LIN {X 0,Y 247.063,Z 768.988,A -85,B 0,C 180,E1 -18816.531,E2 -18816.531} C_VEL
LIN {X 0,Y 247.331,Z 765.214,A -85,B 0,C 180,E1 -18819.814,E2 -18819.814} C_VEL
LIN {X 0,Y 248.197,Z 759.827,A -85,B 0,C 180,E1 -18823.091,E2 -18823.091} C_VEL
LIN {X 0,Y 249.368,Z 753.588,A -85,B 0,C 180,E1 -18825.947,E2 -18825.947} C_VEL
LIN {X 0,Y 251.192,Z 745.733,A -85,B 0,C 180,E1 -18828.767,E2 -18828.767} C_VEL
LIN {X 0,Y 253.14,Z 737.491,A -85,B 0,C 180,E1 -18831.154,E2 -18831.154} C_VEL
LIN {X 0,Y 255.134,Z 729.322,A -85,B 0,C 180,E1 -18833.11,E2 -18833.11} C_VEL
LIN {X 0,Y 257.768,Z 718.537,A -85,B 0,C 180,E1 -18835.212,E2 -18835.212} C_VEL
LIN {X 0,Y 260.138,Z 707.083,A -85,B 0,C 180,E1 -18837.029,E2 -18837.029} C_VEL
LIN {X 0,Y 262.65,Z 694.698,A -85,B 0,C 180,E1 -18838.572,E2 -18838.572} C_VEL
LIN {X 0,Y 264.885,Z 681.638,A -85,B 0,C 180,E1 -18839.831,E2 -18839.831} C_VEL
LIN {X 0,Y 266.701,Z 667.987,A -85,B 0,C 180,E1 -18840.808,E2 -18840.808} C_VEL
LIN {X 0,Y 268.128,Z 653.813,A -85,B 0,C 180,E1 -18841.503,E2 -18841.503} C_VEL
LIN {X 0,Y 269.125,Z 632.659,A -85,B 0,C 180,E1 -18842.143,E2 -18842.143} C_VEL
LIN {X 0,Y 271.804,Z 565.547,A -85,B 0,C 180,E1 -18843.958,E2 -18843.958} C_VEL
LIN {X 0,Y 269.236,Z 545.201,A -85,B 0,C 180,E1 -18844.967,E2 -18844.967} C_VEL
LIN {X 0,Y 261.457,Z 528.213,A -85,B 0,C 180,E1 -18846.671,E2 -18846.671} C_VEL
LIN {X 0,Y 257.903,Z 520.842,A -85,B 0,C 180,E1 -18847.537,E2 -18847.537} C_VEL
LIN {X 0,Y 255.154,Z 510.348,A -85,B 0,C 180,E1 -18851.377,E2 -18851.377} C_VEL
LIN {X 0,Y 252.343,Z 500.973,A -85,B 0,C 180,E1 -18855.158,E2 -18855.158} C_VEL
LIN {X 0,Y 249.727,Z 493.237,A -85,B 0,C 180,E1 -18858.597,E2 -18858.597} C_VEL
LIN {X 0,Y 249.076,Z 491.075,A -85,B 0,C 180,E1 -18859.623,E2 -18859.623} C_VEL
LIN {X 0,Y 249.067,Z 491.051,A -85,B 0,C 180,E1 -18863.661,E2 -18863.661} C_VEL
LIN {X 0,Y 249.031,Z 491.083,A -85,B 0,C 180,E1 -18867.843,E2 -18867.843} C_VEL
LIN {X 0,Y 249.088,Z 491.077,A -85,B 0,C 180,E1 -18871.337,E2 -18871.337} C_VEL
LIN {X 0,Y 249.125,Z 491.073,A -85,B 0,C 180,E1 -18874.966,E2 -18874.966} C_VEL
LIN {X 0,Y 249.083,Z 491.04,A -85,B 0,C 180,E1 -18878.601,E2 -18878.601} C_VEL
LIN {X 0,Y 249.232,Z 491.055,A -85,B 0,C 180,E1 -18883.621,E2 -18883.621} C_VEL
LIN {X 0,Y 249.243,Z 491.051,A -85,B 0,C 180,E1 -18888.616,E2 -18888.616} C_VEL
LIN {X 0,Y 249.474,Z 491.033,A -85,B 0,C 180,E1 -18891.903,E2 -18891.903} C_VEL
LIN {X 0,Y 249.429,Z 491.037,A -85,B 0,C 180,E1 -18896.77,E2 -18896.77} C_VEL
LIN {X 0,Y 249.726,Z 490.999,A -85,B 0,C 180,E1 -18900,E2 -18900} C_VEL
LIN {X 0,Y 249.427,Z 491.025,A -85,B 0,C 180,E1 -18903.231,E2 -18903.231} C_VEL
LIN {X 0,Y 249.471,Z 491.022,A -85,B 0,C 180,E1 -18908.098,E2 -18908.098} C_VEL
LIN {X 0,Y 249.243,Z 491.062,A -85,B 0,C 180,E1 -18911.384,E2 -18911.384} C_VEL
LIN {X 0,Y 249.232,Z 491.062,A -85,B 0,C 180,E1 -18916.379,E2 -18916.379} C_VEL
LIN {X 0,Y 249.078,Z 491.076,A -85,B 0,C 180,E1 -18921.519,E2 -18921.519} C_VEL
LIN {X 0,Y 249.122,Z 491.072,A -85,B 0,C 180,E1 -18925.484,E2 -18925.484} C_VEL
LIN {X 0,Y 249.078,Z 491.081,A -85,B 0,C 180,E1 -18928.996,E2 -18928.996} C_VEL
LIN {X 0,Y 249.029,Z 491.089,A -85,B 0,C 180,E1 -18932.426,E2 -18932.426} C_VEL
LIN {X 0,Y 249.067,Z 491.082,A -85,B 0,C 180,E1 -18936.34,E2 -18936.34} C_VEL
LIN {X 0,Y 249.031,Z 491.085,A -85,B 0,C 180,E1 -18940.474,E2 -18940.474} C_VEL
LIN {X 0,Y 249.035,Z 491.107,A -85,B 0,C 180,E1 -18943.626,E2 -18943.626} C_VEL
LIN {X 0,Y 251.756,Z 499.925,A -85,B 0,C 180,E1 -18947.938,E2 -18947.938} C_VEL
LIN {X 0,Y 254.099,Z 507.969,A -85,B 0,C 180,E1 -18951.512,E2 -18951.512} C_VEL
LIN {X 0,Y 256.491,Z 517.849,A -85,B 0,C 180,E1 -18955.457,E2 -18955.457} C_VEL
LIN {X 0,Y 265.338,Z 535.856,A -85,B 0,C 180,E1 -18957.4,E2 -18957.4} C_VEL
LIN {X 0,Y 268.057,Z 542.537,A -85,B 0,C 180,E1 -18957.996,E2 -18957.996} C_VEL
LIN {X 0,Y 271.456,Z 561.971,A -85,B 0,C 180,E1 -18959.038,E2 -18959.038} C_VEL
LIN {X 0,Y 268.937,Z 634.412,A -85,B 0,C 180,E1 -18960.824,E2 -18960.824} C_VEL
LIN {X 0,Y 268.042,Z 647.399,A -85,B 0,C 180,E1 -18961.414,E2 -18961.414} C_VEL
LIN {X 0,Y 266.613,Z 660.621,A -85,B 0,C 180,E1 -18962.318,E2 -18962.318} C_VEL
LIN {X 0,Y 264.864,Z 672.318,A -85,B 0,C 180,E1 -18963.402,E2 -18963.402} C_VEL
LIN {X 0,Y 262.878,Z 683.019,A -85,B 0,C 180,E1 -18964.677,E2 -18964.677} C_VEL
LIN {X 0,Y 260.529,Z 694.027,A -85,B 0,C 180,E1 -18966.34,E2 -18966.34} C_VEL
LIN {X 0,Y 258.055,Z 704.78,A -85,B 0,C 180,E1 -18968.431,E2 -18968.431} C_VEL
LIN {X 0,Y 255.512,Z 714.223,A -85,B 0,C 180,E1 -18970.73,E2 -18970.73} C_VEL
LIN {X 0,Y 253.385,Z 721.843,A -85,B 0,C 180,E1 -18973.071,E2 -18973.071} C_VEL
LIN {X 0,Y 251.62,Z 728.003,A -85,B 0,C 180,E1 -18975.443,E2 -18975.443} C_VEL
LIN {X 0,Y 250.065,Z 732.962,A -85,B 0,C 180,E1 -18977.834,E2 -18977.834} C_VEL
LIN {X 0,Y 248.951,Z 736.845,A -85,B 0,C 180,E1 -18980.25,E2 -18980.25} C_VEL
LIN {X 0,Y 248.345,Z 739.142,A -85,B 0,C 180,E1 -18982.089,E2 -18982.089} C_VEL
LIN {X 0,Y 247.705,Z 741.812,A -85,B 0,C 180,E1 -18985.119,E2 -18985.119} C_VEL
LIN {X 0,Y 247.294,Z 743.275,A -85,B 0,C 180,E1 -18988.374,E2 -18988.374} C_VEL
LIN {X 0,Y 247.293,Z 743.308,A -85,B 0,C 180,E1 -18991.631,E2 -18991.631} C_VEL
LIN {X 0,Y 247.692,Z 741.889,A -85,B 0,C 180,E1 -18994.885,E2 -18994.885} C_VEL
LIN {X 0,Y 248.44,Z 739.032,A -85,B 0,C 180,E1 -18998.133,E2 -18998.133} C_VEL
LIN {X 0,Y 249.249,Z 735.827,A -85,B 0,C 180,E1 -19000.563,E2 -19000.563} C_VEL
LIN {X 0,Y 250.503,Z 731.638,A -85,B 0,C 180,E1 -19002.972,E2 -19002.972} C_VEL
LIN {X 0,Y 252.36,Z 725.378,A -85,B 0,C 180,E1 -19005.757,E2 -19005.757} C_VEL
LIN {X 0,Y 254.34,Z 718.607,A -85,B 0,C 180,E1 -19008.113,E2 -19008.113} C_VEL
LIN {X 0,Y 256.246,Z 711.743,A -85,B 0,C 180,E1 -19010.052,E2 -19010.052} C_VEL
LIN {X 0,Y 258.424,Z 703.542,A -85,B 0,C 180,E1 -19011.961,E2 -19011.961} C_VEL
LIN {X 0,Y 260.663,Z 693.6,A -85,B 0,C 180,E1 -19013.857,E2 -19013.857} C_VEL
LIN {X 0,Y 263.036,Z 682.426,A -85,B 0,C 180,E1 -19015.523,E2 -19015.523} C_VEL
LIN {X 0,Y 265.334,Z 669.82,A -85,B 0,C 180,E1 -19016.977,E2 -19016.977} C_VEL
LIN {X 0,Y 267.087,Z 657.397,A -85,B 0,C 180,E1 -19018.059,E2 -19018.059} C_VEL
LIN {X 0,Y 268.355,Z 644.28,A -85,B 0,C 180,E1 -19018.874,E2 -19018.874} C_VEL
LIN {X 0,Y 269.273,Z 630.239,A -85,B 0,C 180,E1 -19019.408,E2 -19019.408} C_VEL
LIN {X 0,Y 271.407,Z 561.361,A -85,B 0,C 180,E1 -19021.114,E2 -19021.114} C_VEL
LIN {X 0,Y 267.964,Z 541.862,A -85,B 0,C 180,E1 -19022.167,E2 -19022.167} C_VEL
LIN {X 0,Y 261.576,Z 528.117,A -85,B 0,C 180,E1 -19023.54,E2 -19023.54} C_VEL
LIN {X 0,Y 256.403,Z 517.647,A -85,B 0,C 180,E1 -19024.716,E2 -19024.716} C_VEL
LIN {X 0,Y 254.602,Z 509.943,A -85,B 0,C 180,E1 -19027.81,E2 -19027.81} C_VEL
LIN {X 0,Y 252.374,Z 502.038,A -85,B 0,C 180,E1 -19031.246,E2 -19031.246} C_VEL
LIN {X 0,Y 249.777,Z 493.563,A -85,B 0,C 180,E1 -19035.297,E2 -19035.297} C_VEL
LIN {X 0,Y 249.035,Z 491.083,A -85,B 0,C 180,E1 -19036.66,E2 -19036.66} C_VEL
LIN {X 0,Y 249.014,Z 491.092,A -85,B 0,C 180,E1 -19039.646,E2 -19039.646} C_VEL
LIN {X 0,Y 249.152,Z 491.24,A -85,B 0,C 180,E1 -19043.799,E2 -19043.799} C_VEL
LIN {X 0,Y 253.198,Z 509.007,A -85,B 0,C 180,E1 -19048.171,E2 -19048.171} C_VEL
LIN {X 0,Y 255.988,Z 522.126,A -85,B 0,C 180,E1 -19051.285,E2 -19051.285} C_VEL
LIN {X 0,Y 254.745,Z 535.168,A -85,B 0,C 180,E1 -19054.075,E2 -19054.075} C_VEL
LIN {X 0,Y 256.845,Z 557.306,A -85,B 0,C 180,E1 -19055.19,E2 -19055.19} C_VEL
LIN {X 0,Y 257.538,Z 564.571,A -85,B 0,C 180,E1 -19055.55,E2 -19055.55} C_VEL
LIN {X 0,Y 255.657,Z 605.87,A -85,B 0,C 180,E1 -19057.353,E2 -19057.353} C_VEL
LIN {X 0,Y 254.757,Z 611.621,A -85,B 0,C 180,E1 -19057.58,E2 -19057.58} C_VEL
LIN {X 0,Y 248.289,Z 630.154,A -85,B 0,C 180,E1 -19058.245,E2 -19058.245} C_VEL
LIN {X 0,Y 247.394,Z 635.9,A -85,B 0,C 180,E1 -19058.493,E2 -19058.493} C_VEL
LIN {X 0,Y 246.583,Z 652.231,A -85,B 0,C 180,E1 -19059.347,E2 -19059.347} C_VEL
LIN {X 0,Y 245.788,Z 666.512,A -85,B 0,C 180,E1 -19060.451,E2 -19060.451} C_VEL
LIN {X 0,Y 244.809,Z 679.521,A -85,B 0,C 180,E1 -19061.808,E2 -19061.808} C_VEL
LIN {X 0,Y 243.825,Z 691.891,A -85,B 0,C 180,E1 -19063.463,E2 -19063.463} C_VEL
LIN {X 0,Y 242.795,Z 703.085,A -85,B 0,C 180,E1 -19065.328,E2 -19065.328} C_VEL
LIN {X 0,Y 241.849,Z 713.215,A -85,B 0,C 180,E1 -19067.411,E2 -19067.411} C_VEL
LIN {X 0,Y 241.065,Z 723.166,A -85,B 0,C 180,E1 -19069.926,E2 -19069.926} C_VEL
LIN {X 0,Y 240.487,Z 731.109,A -85,B 0,C 180,E1 -19072.443,E2 -19072.443} C_VEL
LIN {X 0,Y 240.123,Z 737.48,A -85,B 0,C 180,E1 -19074.962,E2 -19074.962} C_VEL
LIN {X 0,Y 240.068,Z 742.54,A -85,B 0,C 180,E1 -19077.483,E2 -19077.483} C_VEL
LIN {X 0,Y 240.001,Z 746.415,A -85,B 0,C 180,E1 -19080,E2 -19080} C_VEL
LIN {X 0,Y 240.132,Z 748.396,A -85,B 0,C 180,E1 -19081.677,E2 -19081.677} C_VEL
LIN {X 0,Y 240.339,Z 749.941,A -85,B 0,C 180,E1 -19083.353,E2 -19083.353} C_VEL
LIN {X 0,Y 240.599,Z 751.071,A -85,B 0,C 180,E1 -19085.027,E2 -19085.027} C_VEL
LIN {X 0,Y 240.986,Z 751.787,A -85,B 0,C 180,E1 -19086.699,E2 -19086.699} C_VEL
LIN {X 0,Y 242.491,Z 751.94,A -85,B 0,C 180,E1 -19090.014,E2 -19090.014} C_VEL
LIN {X 0,Y 243.475,Z 751.426,A -85,B 0,C 180,E1 -19091.657,E2 -19091.657} C_VEL
LIN {X 0,Y 244.569,Z 750.511,A -85,B 0,C 180,E1 -19093.29,E2 -19093.29} C_VEL
LIN {X 0,Y 245.887,Z 749.165,A -85,B 0,C 180,E1 -19094.906,E2 -19094.906} C_VEL
LIN {X 0,Y 248.313,Z 746.344,A -85,B 0,C 180,E1 -19097.288,E2 -19097.288} C_VEL
LIN {X 0,Y 251.19,Z 742.532,A -85,B 0,C 180,E1 -19099.618,E2 -19099.618} C_VEL
LIN {X 0,Y 254.431,Z 737.639,A -85,B 0,C 180,E1 -19101.895,E2 -19101.895} C_VEL
LIN {X 0,Y 258.83,Z 730.384,A -85,B 0,C 180,E1 -19104.461,E2 -19104.461} C_VEL
LIN {X 0,Y 263.038,Z 722.604,A -85,B 0,C 180,E1 -19106.586,E2 -19106.586} C_VEL
LIN {X 0,Y 267.643,Z 713.173,A -85,B 0,C 180,E1 -19108.635,E2 -19108.635} C_VEL
LIN {X 0,Y 271.73,Z 703.612,A -85,B 0,C 180,E1 -19110.288,E2 -19110.288} C_VEL
LIN {X 0,Y 276.114,Z 692.145,A -85,B 0,C 180,E1 -19111.881,E2 -19111.881} C_VEL
LIN {X 0,Y 280.348,Z 679.099,A -85,B 0,C 180,E1 -19113.256,E2 -19113.256} C_VEL
LIN {X 0,Y 283.777,Z 666.49,A -85,B 0,C 180,E1 -19114.293,E2 -19114.293} C_VEL
LIN {X 0,Y 286.875,Z 652.054,A -85,B 0,C 180,E1 -19115.149,E2 -19115.149} C_VEL
LIN {X 0,Y 299.377,Z 586.891,A -85,B 0,C 180,E1 -19118.099,E2 -19118.099} C_VEL
LIN {X 0,Y 299.506,Z 583.69,A -85,B 0,C 180,E1 -19118.593,E2 -19118.593} C_VEL
LIN {X 0,Y 298.716,Z 579.452,A -85,B 0,C 180,E1 -19120.201,E2 -19120.201} C_VEL
LIN {X 0,Y 298.09,Z 576.112,A -85,B 0,C 180,E1 -19122.158,E2 -19122.158} C_VEL
LIN {X 0,Y 297.908,Z 574.347,A -85,B 0,C 180,E1 -19124.166,E2 -19124.166} C_VEL
LIN {X 0,Y 297.981,Z 573.981,A -85,B 0,C 180,E1 -19125.037,E2 -19125.037} C_VEL
LIN {X 0,Y 298.861,Z 574.179,A -85,B 0,C 180,E1 -19127.517,E2 -19127.517} C_VEL
LIN {X 0,Y 299.892,Z 575.224,A -85,B 0,C 180,E1 -19129.089,E2 -19129.089} C_VEL
LIN {X 0,Y 299.897,Z 577.189,A -85,B 0,C 180,E1 -19129.569,E2 -19129.569} C_VEL
LIN {X 0,Y 281.311,Z 668.892,A -85,B 0,C 180,E1 -19133.825,E2 -19133.825} C_VEL
LIN {X 0,Y 277.549,Z 683.549,A -85,B 0,C 180,E1 -19134.824,E2 -19134.824} C_VEL
LIN {X 0,Y 273.49,Z 696.788,A -85,B 0,C 180,E1 -19136.017,E2 -19136.017} C_VEL
LIN {X 0,Y 268.788,Z 709.942,A -85,B 0,C 180,E1 -19137.585,E2 -19137.585} C_VEL
LIN {X 0,Y 264.498,Z 720.789,A -85,B 0,C 180,E1 -19139.235,E2 -19139.235} C_VEL
LIN {X 0,Y 259.933,Z 731.584,A -85,B 0,C 180,E1 -19141.318,E2 -19141.318} C_VEL
LIN {X 0,Y 255.638,Z 740.658,A -85,B 0,C 180,E1 -19143.463,E2 -19143.463} C_VEL
LIN {X 0,Y 251.355,Z 749.308,A -85,B 0,C 180,E1 -19146.08,E2 -19146.08} C_VEL
LIN {X 0,Y 248.314,Z 755.403,A -85,B 0,C 180,E1 -19148.409,E2 -19148.409} C_VEL
LIN {X 0,Y 245.94,Z 759.945,A -85,B 0,C 180,E1 -19150.563,E2 -19150.563} C_VEL
LIN {X 0,Y 243.719,Z 764.366,A -85,B 0,C 180,E1 -19153.238,E2 -19153.238} C_VEL
LIN {X 0,Y 241.577,Z 768.25,A -85,B 0,C 180,E1 -19156.54,E2 -19156.54} C_VEL
LIN {X 0,Y 240.411,Z 770.486,A -85,B 0,C 180,E1 -19159.896,E2 -19159.896} C_VEL
LIN {X 0,Y 239.941,Z 771.177,A -85,B 0,C 180,E1 -19163.27,E2 -19163.27} C_VEL
LIN {X 0,Y 240.025,Z 770.527,A -85,B 0,C 180,E1 -19166.011,E2 -19166.011} C_VEL
LIN {X 0,Y 240.074,Z 771.413,A -85,B 0,C 180,E1 -19168.32,E2 -19168.32} C_VEL
LIN {X 0,Y 240.126,Z 771.603,A -85,B 0,C 180,E1 -19169.998,E2 -19169.998} C_VEL
LIN {X 0,Y 240.072,Z 771.405,A -85,B 0,C 180,E1 -19171.675,E2 -19171.675} C_VEL
LIN {X 0,Y 240.016,Z 770.832,A -85,B 0,C 180,E1 -19173.355,E2 -19173.355} C_VEL
LIN {X 0,Y 239.99,Z 769.684,A -85,B 0,C 180,E1 -19175.331,E2 -19175.331} C_VEL
LIN {X 0,Y 240.106,Z 766.883,A -85,B 0,C 180,E1 -19178.413,E2 -19178.413} C_VEL
LIN {X 0,Y 240.626,Z 762.311,A -85,B 0,C 180,E1 -19181.795,E2 -19181.795} C_VEL
LIN {X 0,Y 241.543,Z 757.744,A -85,B 0,C 180,E1 -19184.316,E2 -19184.316} C_VEL
LIN {X 0,Y 243.018,Z 750.745,A -85,B 0,C 180,E1 -19187.379,E2 -19187.379} C_VEL
LIN {X 0,Y 245.05,Z 742.755,A -85,B 0,C 180,E1 -19190.128,E2 -19190.128} C_VEL
LIN {X 0,Y 247.241,Z 733.954,A -85,B 0,C 180,E1 -19192.563,E2 -19192.563} C_VEL
LIN {X 0,Y 250.045,Z 723.237,A -85,B 0,C 180,E1 -19194.933,E2 -19194.933} C_VEL
LIN {X 0,Y 252.611,Z 711.964,A -85,B 0,C 180,E1 -19196.949,E2 -19196.949} C_VEL
LIN {X 0,Y 255.109,Z 700.402,A -85,B 0,C 180,E1 -19198.596,E2 -19198.596} C_VEL
LIN {X 0,Y 257.705,Z 687.061,A -85,B 0,C 180,E1 -19200.071,E2 -19200.071} C_VEL
LIN {X 0,Y 259.748,Z 674.02,A -85,B 0,C 180,E1 -19201.16,E2 -19201.16} C_VEL
LIN {X 0,Y 261.35,Z 660.795,A -85,B 0,C 180,E1 -19201.964,E2 -19201.964} C_VEL
LIN {X 0,Y 262.518,Z 646.244,A -85,B 0,C 180,E1 -19202.541,E2 -19202.541} C_VEL
LIN {X 0,Y 265.82,Z 566.599,A -85,B 0,C 180,E1 -19204.744,E2 -19204.744} C_VEL
LIN {X 0,Y 263.639,Z 548.18,A -85,B 0,C 180,E1 -19205.672,E2 -19205.672} C_VEL
LIN {X 0,Y 256.348,Z 532.11,A -85,B 0,C 180,E1 -19207.339,E2 -19207.339} C_VEL
LIN {X 0,Y 250.739,Z 520.88,A -85,B 0,C 180,E1 -19208.7,E2 -19208.7} C_VEL
LIN {X 0,Y 248.078,Z 510.843,A -85,B 0,C 180,E1 -19212.56,E2 -19212.56} C_VEL
LIN {X 0,Y 245.221,Z 501.526,A -85,B 0,C 180,E1 -19216.541,E2 -19216.541} C_VEL
LIN {X 0,Y 242.876,Z 494.517,A -85,B 0,C 180,E1 -19219.845,E2 -19219.845} C_VEL
LIN {X 0,Y 241.988,Z 491.961,A -85,B 0,C 180,E1 -19221.217,E2 -19221.217} C_VEL
LIN {X 0,Y 242.028,Z 491.926,A -85,B 0,C 180,E1 -19224.496,E2 -19224.496} C_VEL
LIN {X 0,Y 241.967,Z 491.959,A -85,B 0,C 180,E1 -19228.479,E2 -19228.479} C_VEL
LIN {X 0,Y 241.997,Z 491.957,A -85,B 0,C 180,E1 -19232.312,E2 -19232.312} C_VEL
LIN {X 0,Y 242.031,Z 491.933,A -85,B 0,C 180,E1 -19236.013,E2 -19236.013} C_VEL
LIN {X 0,Y 242.025,Z 491.929,A -85,B 0,C 180,E1 -19239.607,E2 -19239.607} C_VEL
LIN {X 0,Y 242.153,Z 491.939,A -85,B 0,C 180,E1 -19243.278,E2 -19243.278} C_VEL
LIN {X 0,Y 242.177,Z 491.932,A -85,B 0,C 180,E1 -19248.28,E2 -19248.28} C_VEL
LIN {X 0,Y 242.425,Z 491.912,A -85,B 0,C 180,E1 -19251.666,E2 -19251.666} C_VEL
LIN {X 0,Y 242.254,Z 491.928,A -85,B 0,C 180,E1 -19255.007,E2 -19255.007} C_VEL
LIN {X 0,Y 242.628,Z 491.873,A -85,B 0,C 180,E1 -19258.34,E2 -19258.34} C_VEL
LIN {X 0,Y 242.627,Z 491.887,A -85,B 0,C 180,E1 -19261.66,E2 -19261.66} C_VEL
LIN {X 0,Y 242.418,Z 491.91,A -85,B 0,C 180,E1 -19266.744,E2 -19266.744} C_VEL
LIN {X 0,Y 242.304,Z 491.924,A -85,B 0,C 180,E1 -19270.022,E2 -19270.022} C_VEL
LIN {X 0,Y 242.157,Z 491.946,A -85,B 0,C 180,E1 -19275.142,E2 -19275.142} C_VEL
LIN {X 0,Y 242.064,Z 491.947,A -85,B 0,C 180,E1 -19278.625,E2 -19278.625} C_VEL
LIN {X 0,Y 242.004,Z 491.954,A -85,B 0,C 180,E1 -19282.181,E2 -19282.181} C_VEL
LIN {X 0,Y 242.058,Z 491.949,A -85,B 0,C 180,E1 -19285.839,E2 -19285.839} C_VEL
LIN {X 0,Y 242.023,Z 491.955,A -85,B 0,C 180,E1 -19289.581,E2 -19289.581} C_VEL
LIN {X 0,Y 241.984,Z 491.959,A -85,B 0,C 180,E1 -19293.493,E2 -19293.493} C_VEL
LIN {X 0,Y 242.003,Z 491.958,A -85,B 0,C 180,E1 -19297.58,E2 -19297.58} C_VEL
LIN {X 0,Y 242.002,Z 492.051,A -85,B 0,C 180,E1 -19302.172,E2 -19302.172} C_VEL
LIN {X 0,Y 244.563,Z 500.18,A -85,B 0,C 180,E1 -19306.398,E2 -19306.398} C_VEL
LIN {X 0,Y 246.96,Z 508.301,A -85,B 0,C 180,E1 -19310.208,E2 -19310.208} C_VEL
LIN {X 0,Y 249.145,Z 517.089,A -85,B 0,C 180,E1 -19313.965,E2 -19313.965} C_VEL
LIN {X 0,Y 249.339,Z 517.876,A -85,B 0,C 180,E1 -19314.248,E2 -19314.248} C_VEL
LIN {X 0,Y 257.668,Z 534.339,A -85,B 0,C 180,E1 -19316.183,E2 -19316.183} C_VEL
LIN {X 0,Y 262.372,Z 544.96,A -85,B 0,C 180,E1 -19317.243,E2 -19317.243} C_VEL
LIN {X 0,Y 265.482,Z 563.212,A -85,B 0,C 180,E1 -19318.248,E2 -19318.248} C_VEL
LIN {X 0,Y 262.806,Z 635.476,A -85,B 0,C 180,E1 -19320.075,E2 -19320.075} C_VEL
LIN {X 0,Y 261.873,Z 648.172,A -85,B 0,C 180,E1 -19320.676,E2 -19320.676} C_VEL
LIN {X 0,Y 260.362,Z 661.261,A -85,B 0,C 180,E1 -19321.594,E2 -19321.594} C_VEL
LIN {X 0,Y 258.562,Z 672.88,A -85,B 0,C 180,E1 -19322.701,E2 -19322.701} C_VEL
LIN {X 0,Y 256.206,Z 684.892,A -85,B 0,C 180,E1 -19324.187,E2 -19324.187} C_VEL
LIN {X 0,Y 253.796,Z 695.719,A -85,B 0,C 180,E1 -19325.925,E2 -19325.925} C_VEL
LIN {X 0,Y 251.492,Z 705.227,A -85,B 0,C 180,E1 -19327.838,E2 -19327.838} C_VEL
LIN {X 0,Y 248.846,Z 714.658,A -85,B 0,C 180,E1 -19330.192,E2 -19330.192} C_VEL
LIN {X 0,Y 246.626,Z 722.266,A -85,B 0,C 180,E1 -19332.592,E2 -19332.592} C_VEL
LIN {X 0,Y 244.754,Z 728.421,A -85,B 0,C 180,E1 -19335.025,E2 -19335.025} C_VEL
LIN {X 0,Y 243.132,Z 733.378,A -85,B 0,C 180,E1 -19337.481,E2 -19337.481} C_VEL
LIN {X 0,Y 241.965,Z 737.258,A -85,B 0,C 180,E1 -19339.966,E2 -19339.966} C_VEL
LIN {X 0,Y 241.269,Z 739.756,A -85,B 0,C 180,E1 -19342.056,E2 -19342.056} C_VEL
LIN {X 0,Y 240.662,Z 742.221,A -85,B 0,C 180,E1 -19344.976,E2 -19344.976} C_VEL
LIN {X 0,Y 240.219,Z 743.683,A -85,B 0,C 180,E1 -19348.326,E2 -19348.326} C_VEL
LIN {X 0,Y 240.218,Z 743.716,A -85,B 0,C 180,E1 -19351.679,E2 -19351.679} C_VEL
LIN {X 0,Y 240.648,Z 742.297,A -85,B 0,C 180,E1 -19355.028,E2 -19355.028} C_VEL
LIN {X 0,Y 241.435,Z 739.44,A -85,B 0,C 180,E1 -19358.371,E2 -19358.371} C_VEL
LIN {X 0,Y 242.296,Z 736.237,A -85,B 0,C 180,E1 -19360.87,E2 -19360.87} C_VEL
LIN {X 0,Y 243.608,Z 732.051,A -85,B 0,C 180,E1 -19363.346,E2 -19363.346} C_VEL
LIN {X 0,Y 245.552,Z 725.793,A -85,B 0,C 180,E1 -19366.206,E2 -19366.206} C_VEL
LIN {X 0,Y 247.596,Z 719.03,A -85,B 0,C 180,E1 -19368.625,E2 -19368.625} C_VEL
LIN {X 0,Y 250.107,Z 710.653,A -85,B 0,C 180,E1 -19370.996,E2 -19370.996} C_VEL
LIN {X 0,Y 252.615,Z 701.132,A -85,B 0,C 180,E1 -19373.155,E2 -19373.155} C_VEL
LIN {X 0,Y 254.962,Z 690.605,A -85,B 0,C 180,E1 -19375.077,E2 -19375.077} C_VEL
LIN {X 0,Y 257.31,Z 680.098,A -85,B 0,C 180,E1 -19376.57,E2 -19376.57} C_VEL
LIN {X 0,Y 259.371,Z 668.588,A -85,B 0,C 180,E1 -19377.868,E2 -19377.868} C_VEL
LIN {X 0,Y 261.169,Z 655.482,A -85,B 0,C 180,E1 -19378.974,E2 -19378.974} C_VEL
LIN {X 0,Y 262.464,Z 642.331,A -85,B 0,C 180,E1 -19379.752,E2 -19379.752} C_VEL
LIN {X 0,Y 263.237,Z 629.949,A -85,B 0,C 180,E1 -19380.207,E2 -19380.207} C_VEL
LIN {X 0,Y 265.415,Z 562.327,A -85,B 0,C 180,E1 -19381.917,E2 -19381.917} C_VEL
LIN {X 0,Y 262.191,Z 544.284,A -85,B 0,C 180,E1 -19382.939,E2 -19382.939} C_VEL
LIN {X 0,Y 254.799,Z 528.512,A -85,B 0,C 180,E1 -19384.606,E2 -19384.606} C_VEL
LIN {X 0,Y 249.291,Z 517.693,A -85,B 0,C 180,E1 -19385.939,E2 -19385.939} C_VEL
LIN {X 0,Y 247.457,Z 510.196,A -85,B 0,C 180,E1 -19389.105,E2 -19389.105} C_VEL
LIN {X 0,Y 245.027,Z 501.746,A -85,B 0,C 180,E1 -19392.996,E2 -19392.996} C_VEL
LIN {X 0,Y 242.652,Z 494.199,A -85,B 0,C 180,E1 -19396.844,E2 -19396.844} C_VEL
LIN {X 0,Y 241.945,Z 491.959,A -85,B 0,C 180,E1 -19398.079,E2 -19398.079} C_VEL
LIN {X 0,Y 242.004,Z 491.948,A -85,B 0,C 180,E1 -19402.42,E2 -19402.42} C_VEL
LIN {X 0,Y 242.065,Z 492.11,A -85,B 0,C 180,E1 -19403.398,E2 -19403.398} C_VEL
LIN {X 0,Y 245.421,Z 506.589,A -85,B 0,C 180,E1 -19407.037,E2 -19407.037} C_VEL
LIN {X 0,Y 248.594,Z 521.009,A -85,B 0,C 180,E1 -19410.559,E2 -19410.559} C_VEL
LIN {X 0,Y 249.003,Z 523.045,A -85,B 0,C 180,E1 -19411.044,E2 -19411.044} C_VEL
LIN {X 0,Y 247.813,Z 535.718,A -85,B 0,C 180,E1 -19413.764,E2 -19413.764} C_VEL
LIN {X 0,Y 249.853,Z 558.097,A -85,B 0,C 180,E1 -19414.92,E2 -19414.92} C_VEL
LIN {X 0,Y 250.524,Z 565.139,A -85,B 0,C 180,E1 -19415.281,E2 -19415.281} C_VEL
LIN {X 0,Y 247.394,Z 635.9,A -85,B 0,C 180,E1 -19418.493,E2 -19418.493} C_VEL
LIN {X 0,Y 246.452,Z 641.623,A -85,B 0,C 180,E1 -19418.743,E2 -19418.743} C_VEL
LIN {X 0,Y 243.145,Z 650.765,A -85,B 0,C 180,E1 -19419.191,E2 -19419.191} C_VEL
LIN {X 0,Y 239.816,Z 659.772,A -85,B 0,C 180,E1 -19419.787,E2 -19419.787} C_VEL
LIN {X 0,Y 238.792,Z 665.286,A -85,B 0,C 180,E1 -19420.246,E2 -19420.246} C_VEL
LIN {X 0,Y 237.912,Z 677.304,A -85,B 0,C 180,E1 -19421.484,E2 -19421.484} C_VEL
LIN {X 0,Y 236.892,Z 690.249,A -85,B 0,C 180,E1 -19423.186,E2 -19423.186} C_VEL
LIN {X 0,Y 235.826,Z 701.775,A -85,B 0,C 180,E1 -19425.105,E2 -19425.105} C_VEL
LIN {X 0,Y 234.903,Z 711.285,A -85,B 0,C 180,E1 -19427.033,E2 -19427.033} C_VEL
LIN {X 0,Y 234.19,Z 720.07,A -85,B 0,C 180,E1 -19429.189,E2 -19429.189} C_VEL
LIN {X 0,Y 233.546,Z 728.631,A -85,B 0,C 180,E1 -19431.782,E2 -19431.782} C_VEL
LIN {X 0,Y 233.195,Z 734.723,A -85,B 0,C 180,E1 -19434.032,E2 -19434.032} C_VEL
LIN {X 0,Y 233.008,Z 740.278,A -85,B 0,C 180,E1 -19436.541,E2 -19436.541} C_VEL
LIN {X 0,Y 232.92,Z 744.8,A -85,B 0,C 180,E1 -19439.135,E2 -19439.135} C_VEL
LIN {X 0,Y 233.064,Z 748.185,A -85,B 0,C 180,E1 -19441.728,E2 -19441.728} C_VEL
LIN {X 0,Y 233.259,Z 749.889,A -85,B 0,C 180,E1 -19443.454,E2 -19443.454} C_VEL
LIN {X 0,Y 233.945,Z 752.006,A -85,B 0,C 180,E1 -19446.901,E2 -19446.901} C_VEL
LIN {X 0,Y 235.072,Z 752.52,A -85,B 0,C 180,E1 -19449.377,E2 -19449.377} C_VEL
LIN {X 0,Y 236.569,Z 752.14,A -85,B 0,C 180,E1 -19452.002,E2 -19452.002} C_VEL
LIN {X 0,Y 239.112,Z 750.237,A -85,B 0,C 180,E1 -19455.339,E2 -19455.339} C_VEL
LIN {X 0,Y 240.815,Z 748.652,A -85,B 0,C 180,E1 -19456.968,E2 -19456.968} C_VEL
LIN {X 0,Y 243.622,Z 745.506,A -85,B 0,C 180,E1 -19459.375,E2 -19459.375} C_VEL
LIN {X 0,Y 248.11,Z 739.66,A -85,B 0,C 180,E1 -19462.482,E2 -19462.482} C_VEL
LIN {X 0,Y 252.031,Z 733.958,A -85,B 0,C 180,E1 -19464.726,E2 -19464.726} C_VEL
LIN {X 0,Y 257.149,Z 725.612,A -85,B 0,C 180,E1 -19467.244,E2 -19467.244} C_VEL
LIN {X 0,Y 261.904,Z 716.792,A -85,B 0,C 180,E1 -19469.322,E2 -19469.322} C_VEL
LIN {X 0,Y 266.196,Z 707.988,A -85,B 0,C 180,E1 -19470.986,E2 -19470.986} C_VEL
LIN {X 0,Y 271.215,Z 696.243,A -85,B 0,C 180,E1 -19472.747,E2 -19472.747} C_VEL
LIN {X 0,Y 275.618,Z 684.358,A -85,B 0,C 180,E1 -19474.123,E2 -19474.123} C_VEL
LIN {X 0,Y 279.719,Z 671.098,A -85,B 0,C 180,E1 -19475.301,E2 -19475.301} C_VEL
LIN {X 0,Y 283.08,Z 657.763,A -85,B 0,C 180,E1 -19476.186,E2 -19476.186} C_VEL
LIN {X 0,Y 297.061,Z 589.261,A -85,B 0,C 180,E1 -19479.357,E2 -19479.357} C_VEL
LIN {X 0,Y 296.93,Z 587.865,A -85,B 0,C 180,E1 -19479.797,E2 -19479.797} C_VEL
LIN {X 0,Y 296.438,Z 584.785,A -85,B 0,C 180,E1 -19481.222,E2 -19481.222} C_VEL
LIN {X 0,Y 296.183,Z 582.554,A -85,B 0,C 180,E1 -19482.641,E2 -19482.641} C_VEL
LIN {X 0,Y 296.134,Z 581.054,A -85,B 0,C 180,E1 -19484.602,E2 -19484.602} C_VEL
LIN {X 0,Y 296.925,Z 580.953,A -85,B 0,C 180,E1 -19487.201,E2 -19487.201} C_VEL
LIN {X 0,Y 297.618,Z 581.538,A -85,B 0,C 180,E1 -19488.392,E2 -19488.392} C_VEL
LIN {X 0,Y 278.815,Z 668.546,A -85,B 0,C 180,E1 -19492.431,E2 -19492.431} C_VEL
LIN {X 0,Y 274.544,Z 683.906,A -85,B 0,C 180,E1 -19493.473,E2 -19493.473} C_VEL
LIN {X 0,Y 269.683,Z 698.183,A -85,B 0,C 180,E1 -19494.787,E2 -19494.787} C_VEL
LIN {X 0,Y 264.714,Z 710.91,A -85,B 0,C 180,E1 -19496.341,E2 -19496.341} C_VEL
LIN {X 0,Y 259.678,Z 722.319,A -85,B 0,C 180,E1 -19498.144,E2 -19498.144} C_VEL
LIN {X 0,Y 254.831,Z 732.672,A -85,B 0,C 180,E1 -19500.234,E2 -19500.234} C_VEL
LIN {X 0,Y 249.543,Z 742.705,A -85,B 0,C 180,E1 -19502.762,E2 -19502.762} C_VEL
LIN {X 0,Y 245.037,Z 750.817,A -85,B 0,C 180,E1 -19505.423,E2 -19505.423} C_VEL
LIN {X 0,Y 241.81,Z 756.496,A -85,B 0,C 180,E1 -19507.798,E2 -19507.798} C_VEL
LIN {X 0,Y 238.272,Z 762.492,A -85,B 0,C 180,E1 -19511.065,E2 -19511.065} C_VEL
LIN {X 0,Y 235.708,Z 766.773,A -85,B 0,C 180,E1 -19514.432,E2 -19514.432} C_VEL
LIN {X 0,Y 233.903,Z 769.492,A -85,B 0,C 180,E1 -19517.856,E2 -19517.856} C_VEL
LIN {X 0,Y 233.398,Z 770.291,A -85,B 0,C 180,E1 -19519.589,E2 -19519.589} C_VEL
LIN {X 0,Y 233.056,Z 770.672,A -85,B 0,C 180,E1 -19521.326,E2 -19521.326} C_VEL
LIN {X 0,Y 232.901,Z 770.233,A -85,B 0,C 180,E1 -19524.804,E2 -19524.804} C_VEL
LIN {X 0,Y 232.972,Z 770.006,A -85,B 0,C 180,E1 -19525.66,E2 -19525.66} C_VEL
LIN {X 0,Y 233,Z 771.005,A -85,B 0,C 180,E1 -19528.269,E2 -19528.269} C_VEL
LIN {X 0,Y 233.049,Z 771.195,A -85,B 0,C 180,E1 -19529.998,E2 -19529.998} C_VEL
LIN {X 0,Y 232.997,Z 770.996,A -85,B 0,C 180,E1 -19531.726,E2 -19531.726} C_VEL
LIN {X 0,Y 232.919,Z 769.48,A -85,B 0,C 180,E1 -19535.191,E2 -19535.191} C_VEL
LIN {X 0,Y 233.039,Z 766.469,A -85,B 0,C 180,E1 -19538.67,E2 -19538.67} C_VEL
LIN {X 0,Y 233.624,Z 761.894,A -85,B 0,C 180,E1 -19542.154,E2 -19542.154} C_VEL
LIN {X 0,Y 234.603,Z 757.322,A -85,B 0,C 180,E1 -19544.749,E2 -19544.749} C_VEL
LIN {X 0,Y 236.04,Z 750.862,A -85,B 0,C 180,E1 -19547.677,E2 -19547.677} C_VEL
LIN {X 0,Y 237.972,Z 743.599,A -85,B 0,C 180,E1 -19550.302,E2 -19550.302} C_VEL
LIN {X 0,Y 240.222,Z 735.084,A -85,B 0,C 180,E1 -19552.805,E2 -19552.805} C_VEL
LIN {X 0,Y 243.06,Z 724.757,A -85,B 0,C 180,E1 -19555.242,E2 -19555.242} C_VEL
LIN {X 0,Y 245.629,Z 714.248,A -85,B 0,C 180,E1 -19557.242,E2 -19557.242} C_VEL
LIN {X 0,Y 248.263,Z 702.763,A -85,B 0,C 180,E1 -19558.996,E2 -19558.996} C_VEL
LIN {X 0,Y 250.884,Z 690.115,A -85,B 0,C 180,E1 -19560.51,E2 -19560.51} C_VEL
LIN {X 0,Y 253.167,Z 676.98,A -85,B 0,C 180,E1 -19561.713,E2 -19561.713} C_VEL
LIN {X 0,Y 254.994,Z 663.453,A -85,B 0,C 180,E1 -19562.624,E2 -19562.624} C_VEL
LIN {X 0,Y 256.294,Z 649.35,A -85,B 0,C 180,E1 -19563.257,E2 -19563.257} C_VEL
LIN {X 0,Y 259.922,Z 568.016,A -85,B 0,C 180,E1 -19565.548,E2 -19565.548} C_VEL
LIN {X 0,Y 257.856,Z 550.685,A -85,B 0,C 180,E1 -19566.458,E2 -19566.458} C_VEL
LIN {X 0,Y 251.039,Z 535.558,A -85,B 0,C 180,E1 -19568.091,E2 -19568.091} C_VEL
LIN {X 0,Y 245.079,Z 523.966,A -85,B 0,C 180,E1 -19569.563,E2 -19569.563} C_VEL
LIN {X 0,Y 243.569,Z 520.782,A -85,B 0,C 180,E1 -19569.998,E2 -19569.998} C_VEL
LIN {X 0,Y 240.942,Z 511.185,A -85,B 0,C 180,E1 -19573.909,E2 -19573.909} C_VEL
LIN {X 0,Y 238.042,Z 501.826,A -85,B 0,C 180,E1 -19578.16,E2 -19578.16} C_VEL
LIN {X 0,Y 234.942,Z 492.815,A -85,B 0,C 180,E1 -19582.852,E2 -19582.852} C_VEL
LIN {X 0,Y 234.951,Z 492.839,A -85,B 0,C 180,E1 -19587.424,E2 -19587.424} C_VEL
LIN {X 0,Y 234.941,Z 492.838,A -85,B 0,C 180,E1 -19591.405,E2 -19591.405} C_VEL
LIN {X 0,Y 234.968,Z 492.827,A -85,B 0,C 180,E1 -19595.245,E2 -19595.245} C_VEL
LIN {X 0,Y 234.988,Z 492.796,A -85,B 0,C 180,E1 -19598.968,E2 -19598.968} C_VEL
LIN {X 0,Y 235.086,Z 492.821,A -85,B 0,C 180,E1 -19603.059,E2 -19603.059} C_VEL
LIN {X 0,Y 235.137,Z 492.811,A -85,B 0,C 180,E1 -19607.923,E2 -19607.923} C_VEL
LIN {X 0,Y 235.38,Z 492.79,A -85,B 0,C 180,E1 -19611.414,E2 -19611.414} C_VEL
LIN {X 0,Y 235.396,Z 492.773,A -85,B 0,C 180,E1 -19613.141,E2 -19613.141} C_VEL
LIN {X 0,Y 235.587,Z 492.75,A -85,B 0,C 180,E1 -19618.291,E2 -19618.291} C_VEL
LIN {X 0,Y 235.587,Z 492.763,A -85,B 0,C 180,E1 -19621.71,E2 -19621.71} C_VEL
LIN {X 0,Y 235.394,Z 492.784,A -85,B 0,C 180,E1 -19626.859,E2 -19626.859} C_VEL
LIN {X 0,Y 235.228,Z 492.807,A -85,B 0,C 180,E1 -19630.327,E2 -19630.327} C_VEL
LIN {X 0,Y 235.104,Z 492.825,A -85,B 0,C 180,E1 -19635.607,E2 -19635.607} C_VEL
LIN {X 0,Y 235,Z 492.832,A -85,B 0,C 180,E1 -19639.207,E2 -19639.207} C_VEL
LIN {X 0,Y 234.952,Z 492.834,A -85,B 0,C 180,E1 -19642.884,E2 -19642.884} C_VEL
LIN {X 0,Y 234.962,Z 492.832,A -85,B 0,C 180,E1 -19646.659,E2 -19646.659} C_VEL
LIN {X 0,Y 234.925,Z 492.837,A -85,B 0,C 180,E1 -19650.569,E2 -19650.569} C_VEL
LIN {X 0,Y 234.953,Z 492.837,A -85,B 0,C 180,E1 -19654.635,E2 -19654.635} C_VEL
LIN {X 0,Y 234.935,Z 492.848,A -85,B 0,C 180,E1 -19658.946,E2 -19658.946} C_VEL
LIN {X 0,Y 234.951,Z 493.014,A -85,B 0,C 180,E1 -19660.587,E2 -19660.587} C_VEL
LIN {X 0,Y 237.328,Z 500.443,A -85,B 0,C 180,E1 -19664.711,E2 -19664.711} C_VEL
LIN {X 0,Y 239.575,Z 507.828,A -85,B 0,C 180,E1 -19668.421,E2 -19668.421} C_VEL
LIN {X 0,Y 241.555,Z 515.14,A -85,B 0,C 180,E1 -19671.773,E2 -19671.773} C_VEL
LIN {X 0,Y 242.198,Z 517.803,A -85,B 0,C 180,E1 -19672.933,E2 -19672.933} C_VEL
LIN {X 0,Y 250.66,Z 534.169,A -85,B 0,C 180,E1 -19675.029,E2 -19675.029} C_VEL
LIN {X 0,Y 256.806,Z 547.829,A -85,B 0,C 180,E1 -19676.482,E2 -19676.482} C_VEL
LIN {X 0,Y 259.539,Z 564.051,A -85,B 0,C 180,E1 -19677.409,E2 -19677.409} C_VEL
LIN {X 0,Y 256.79,Z 635.351,A -85,B 0,C 180,E1 -19679.242,E2 -19679.242} C_VEL
LIN {X 0,Y 255.837,Z 648.172,A -85,B 0,C 180,E1 -19679.857,E2 -19679.857} C_VEL
LIN {X 0,Y 254.345,Z 660.766,A -85,B 0,C 180,E1 -19680.745,E2 -19680.745} C_VEL
LIN {X 0,Y 252.292,Z 673.442,A -85,B 0,C 180,E1 -19681.963,E2 -19681.963} C_VEL
LIN {X 0,Y 249.873,Z 685.385,A -85,B 0,C 180,E1 -19683.483,E2 -19683.483} C_VEL
LIN {X 0,Y 247.301,Z 696.379,A -85,B 0,C 180,E1 -19685.292,E2 -19685.292} C_VEL
LIN {X 0,Y 244.956,Z 705.675,A -85,B 0,C 180,E1 -19687.214,E2 -19687.214} C_VEL
LIN {X 0,Y 242.199,Z 715.093,A -85,B 0,C 180,E1 -19689.625,E2 -19689.625} C_VEL
LIN {X 0,Y 239.87,Z 722.69,A -85,B 0,C 180,E1 -19692.085,E2 -19692.085} C_VEL
LIN {X 0,Y 237.913,Z 728.838,A -85,B 0,C 180,E1 -19694.584,E2 -19694.584} C_VEL
LIN {X 0,Y 236.221,Z 733.792,A -85,B 0,C 180,E1 -19697.109,E2 -19697.109} C_VEL
LIN {X 0,Y 234.976,Z 737.672,A -85,B 0,C 180,E1 -19699.664,E2 -19699.664} C_VEL
LIN {X 0,Y 234.178,Z 740.397,A -85,B 0,C 180,E1 -19702.048,E2 -19702.048} C_VEL
LIN {X 0,Y 233.62,Z 742.629,A -85,B 0,C 180,E1 -19704.824,E2 -19704.824} C_VEL
LIN {X 0,Y 233.146,Z 744.092,A -85,B 0,C 180,E1 -19708.275,E2 -19708.275} C_VEL
LIN {X 0,Y 233.145,Z 744.125,A -85,B 0,C 180,E1 -19711.73,E2 -19711.73} C_VEL
LIN {X 0,Y 233.607,Z 742.705,A -85,B 0,C 180,E1 -19715.18,E2 -19715.18} C_VEL
LIN {X 0,Y 234.42,Z 739.849,A -85,B 0,C 180,E1 -19718.623,E2 -19718.623} C_VEL
LIN {X 0,Y 235.341,Z 736.648,A -85,B 0,C 180,E1 -19721.195,E2 -19721.195} C_VEL
LIN {X 0,Y 236.731,Z 732.463,A -85,B 0,C 180,E1 -19723.741,E2 -19723.741} C_VEL
LIN {X 0,Y 238.741,Z 726.21,A -85,B 0,C 180,E1 -19726.682,E2 -19726.682} C_VEL
LIN {X 0,Y 240.89,Z 719.452,A -85,B 0,C 180,E1 -19729.163,E2 -19729.163} C_VEL
LIN {X 0,Y 243.506,Z 711.09,A -85,B 0,C 180,E1 -19731.594,E2 -19731.594} C_VEL
LIN {X 0,Y 246.185,Z 701.231,A -85,B 0,C 180,E1 -19733.879,E2 -19733.879} C_VEL
LIN {X 0,Y 248.584,Z 691.076,A -85,B 0,C 180,E1 -19735.767,E2 -19735.767} C_VEL
LIN {X 0,Y 251.013,Z 680.6,A -85,B 0,C 180,E1 -19737.291,E2 -19737.291} C_VEL
LIN {X 0,Y 253.149,Z 669.152,A -85,B 0,C 180,E1 -19738.616,E2 -19738.616} C_VEL
LIN {X 0,Y 255.027,Z 656.158,A -85,B 0,C 180,E1 -19739.741,E2 -19739.741} C_VEL
LIN {X 0,Y 256.35,Z 643.19,A -85,B 0,C 180,E1 -19740.536,E2 -19740.536} C_VEL
LIN {X 0,Y 257.247,Z 629.661,A -85,B 0,C 180,E1 -19741.044,E2 -19741.044} C_VEL
LIN {X 0,Y 259.535,Z 563.625,A -85,B 0,C 180,E1 -19742.738,E2 -19742.738} C_VEL
LIN {X 0,Y 256.646,Z 547.27,A -85,B 0,C 180,E1 -19743.698,E2 -19743.698} C_VEL
LIN {X 0,Y 249.874,Z 532.638,A -85,B 0,C 180,E1 -19745.296,E2 -19745.296} C_VEL
LIN {X 0,Y 243.458,Z 520.483,A -85,B 0,C 180,E1 -19746.869,E2 -19746.869} C_VEL
LIN {X 0,Y 242.218,Z 517.817,A -85,B 0,C 180,E1 -19747.208,E2 -19747.208} C_VEL
LIN {X 0,Y 239.978,Z 509.276,A -85,B 0,C 180,E1 -19751.052,E2 -19751.052} C_VEL
LIN {X 0,Y 237.432,Z 500.792,A -85,B 0,C 180,E1 -19755.27,E2 -19755.27} C_VEL
LIN {X 0,Y 235.752,Z 495.437,A -85,B 0,C 180,E1 -19758.185,E2 -19758.185} C_VEL
LIN {X 0,Y 234.899,Z 492.851,A -85,B 0,C 180,E1 -19759.684,E2 -19759.684} C_VEL
LIN {X 0,Y 235.014,Z 493.001,A -85,B 0,C 180,E1 -19762.998,E2 -19762.998} C_VEL
LIN {X 0,Y 238.308,Z 507.191,A -85,B 0,C 180,E1 -19766.634,E2 -19766.634} C_VEL
LIN {X 0,Y 241.648,Z 522.216,A -85,B 0,C 180,E1 -19770.368,E2 -19770.368} C_VEL
LIN {X 0,Y 242.019,Z 524.649,A -85,B 0,C 180,E1 -19770.949,E2 -19770.949} C_VEL
LIN {X 0,Y 240.867,Z 535.721,A -85,B 0,C 180,E1 -19773.403,E2 -19773.403} C_VEL
LIN {X 0,Y 242.987,Z 559.548,A -85,B 0,C 180,E1 -19774.673,E2 -19774.673} C_VEL
LIN {X 0,Y 243.588,Z 564.917,A -85,B 0,C 180,E1 -19774.961,E2 -19774.961} C_VEL
LIN {X 0,Y 239.752,Z 648.787,A -85,B 0,C 180,E1 -19779.011,E2 -19779.011} C_VEL
LIN {X 0,Y 238.983,Z 662.691,A -85,B 0,C 180,E1 -19780.02,E2 -19780.02} C_VEL
LIN {X 0,Y 238.792,Z 665.286,A -85,B 0,C 180,E1 -19780.246,E2 -19780.246} C_VEL
LIN {X 0,Y 237.688,Z 670.714,A -85,B 0,C 180,E1 -19780.744,E2 -19780.744} C_VEL
LIN {X 0,Y 234.16,Z 679.206,A -85,B 0,C 180,E1 -19781.651,E2 -19781.651} C_VEL
LIN {X 0,Y 230.635,Z 687.389,A -85,B 0,C 180,E1 -19782.735,E2 -19782.735} C_VEL
LIN {X 0,Y 229.548,Z 692.336,A -85,B 0,C 180,E1 -19783.499,E2 -19783.499} C_VEL
LIN {X 0,Y 228.477,Z 703.732,A -85,B 0,C 180,E1 -19785.527,E2 -19785.527} C_VEL
LIN {X 0,Y 227.52,Z 714.742,A -85,B 0,C 180,E1 -19787.965,E2 -19787.965} C_VEL
LIN {X 0,Y 226.86,Z 722.989,A -85,B 0,C 180,E1 -19790.189,E2 -19790.189} C_VEL
LIN {X 0,Y 226.289,Z 731.099,A -85,B 0,C 180,E1 -19792.863,E2 -19792.863} C_VEL
LIN {X 0,Y 225.98,Z 738.148,A -85,B 0,C 180,E1 -19795.778,E2 -19795.778} C_VEL
LIN {X 0,Y 225.899,Z 742.783,A -85,B 0,C 180,E1 -19798.217,E2 -19798.217} C_VEL
LIN {X 0,Y 225.902,Z 746.772,A -85,B 0,C 180,E1 -19800.891,E2 -19800.891} C_VEL
LIN {X 0,Y 226.181,Z 749.729,A -85,B 0,C 180,E1 -19803.563,E2 -19803.563} C_VEL
LIN {X 0,Y 226.449,Z 751.183,A -85,B 0,C 180,E1 -19805.342,E2 -19805.342} C_VEL
LIN {X 0,Y 226.91,Z 752.191,A -85,B 0,C 180,E1 -19807.116,E2 -19807.116} C_VEL
LIN {X 0,Y 228.569,Z 753,A -85,B 0,C 180,E1 -19810.631,E2 -19810.631} C_VEL
LIN {X 0,Y 229.655,Z 752.825,A -85,B 0,C 180,E1 -19812.369,E2 -19812.369} C_VEL
LIN {X 0,Y 232.345,Z 751.261,A -85,B 0,C 180,E1 -19815.797,E2 -19815.797} C_VEL
LIN {X 0,Y 236.034,Z 748.079,A -85,B 0,C 180,E1 -19819.119,E2 -19819.119} C_VEL
LIN {X 0,Y 239.388,Z 744.566,A -85,B 0,C 180,E1 -19821.529,E2 -19821.529} C_VEL
LIN {X 0,Y 243.115,Z 740.01,A -85,B 0,C 180,E1 -19823.873,E2 -19823.873} C_VEL
LIN {X 0,Y 248.117,Z 733.245,A -85,B 0,C 180,E1 -19826.495,E2 -19826.495} C_VEL
LIN {X 0,Y 253.7,Z 724.705,A -85,B 0,C 180,E1 -19828.998,E2 -19828.998} C_VEL
LIN {X 0,Y 258.888,Z 715.616,A -85,B 0,C 180,E1 -19831.05,E2 -19831.05} C_VEL
LIN {X 0,Y 264.012,Z 705.617,A -85,B 0,C 180,E1 -19832.846,E2 -19832.846} C_VEL
LIN {X 0,Y 269.404,Z 693.334,A -85,B 0,C 180,E1 -19834.569,E2 -19834.569} C_VEL
LIN {X 0,Y 274.18,Z 680.685,A -85,B 0,C 180,E1 -19835.898,E2 -19835.898} C_VEL
LIN {X 0,Y 278.268,Z 667.471,A -85,B 0,C 180,E1 -19836.971,E2 -19836.971} C_VEL
LIN {X 0,Y 281.692,Z 653.632,A -85,B 0,C 180,E1 -19837.793,E2 -19837.793} C_VEL
LIN {X 0,Y 294.699,Z 593.582,A -85,B 0,C 180,E1 -19840.51,E2 -19840.51} C_VEL
LIN {X 0,Y 294.376,Z 590.117,A -85,B 0,C 180,E1 -19842.258,E2 -19842.258} C_VEL
LIN {X 0,Y 294.291,Z 588.286,A -85,B 0,C 180,E1 -19844.039,E2 -19844.039} C_VEL
LIN {X 0,Y 294.549,Z 587.678,A -85,B 0,C 180,E1 -19845.709,E2 -19845.709} C_VEL
LIN {X 0,Y 295.16,Z 587.875,A -85,B 0,C 180,E1 -19847.295,E2 -19847.295} C_VEL
LIN {X 0,Y 277.235,Z 666.329,A -85,B 0,C 180,E1 -19850.904,E2 -19850.904} C_VEL
LIN {X 0,Y 272.983,Z 681.057,A -85,B 0,C 180,E1 -19851.836,E2 -19851.836} C_VEL
LIN {X 0,Y 268.932,Z 692.665,A -85,B 0,C 180,E1 -19852.818,E2 -19852.818} C_VEL
LIN {X 0,Y 263.926,Z 705.052,A -85,B 0,C 180,E1 -19854.136,E2 -19854.136} C_VEL
LIN {X 0,Y 258.825,Z 716.25,A -85,B 0,C 180,E1 -19855.704,E2 -19855.704} C_VEL
LIN {X 0,Y 254.123,Z 725.764,A -85,B 0,C 180,E1 -19857.363,E2 -19857.363} C_VEL
LIN {X 0,Y 248.197,Z 736.798,A -85,B 0,C 180,E1 -19859.825,E2 -19859.825} C_VEL
LIN {X 0,Y 243.491,Z 744.667,A -85,B 0,C 180,E1 -19862.026,E2 -19862.026} C_VEL
LIN {X 0,Y 238.743,Z 752.301,A -85,B 0,C 180,E1 -19864.73,E2 -19864.73} C_VEL
LIN {X 0,Y 234.311,Z 759.105,A -85,B 0,C 180,E1 -19867.978,E2 -19867.978} C_VEL
LIN {X 0,Y 231.576,Z 763.082,A -85,B 0,C 180,E1 -19870.496,E2 -19870.496} C_VEL
LIN {X 0,Y 228.863,Z 767.011,A -85,B 0,C 180,E1 -19873.954,E2 -19873.954} C_VEL
LIN {X 0,Y 227.75,Z 768.397,A -85,B 0,C 180,E1 -19875.706,E2 -19875.706} C_VEL
LIN {X 0,Y 226.382,Z 769.992,A -85,B 0,C 180,E1 -19879.263,E2 -19879.263} C_VEL
LIN {X 0,Y 225.831,Z 770.078,A -85,B 0,C 180,E1 -19882.847,E2 -19882.847} C_VEL
LIN {X 0,Y 225.883,Z 769.355,A -85,B 0,C 180,E1 -19885.044,E2 -19885.044} C_VEL
LIN {X 0,Y 225.927,Z 770.597,A -85,B 0,C 180,E1 -19888.215,E2 -19888.215} C_VEL
LIN {X 0,Y 225.974,Z 770.787,A -85,B 0,C 180,E1 -19889.998,E2 -19889.998} C_VEL
LIN {X 0,Y 225.923,Z 770.587,A -85,B 0,C 180,E1 -19891.78,E2 -19891.78} C_VEL
LIN {X 0,Y 225.84,Z 769.069,A -85,B 0,C 180,E1 -19895.354,E2 -19895.354} C_VEL
LIN {X 0,Y 225.97,Z 766.054,A -85,B 0,C 180,E1 -19898.944,E2 -19898.944} C_VEL
LIN {X 0,Y 226.628,Z 761.477,A -85,B 0,C 180,E1 -19902.535,E2 -19902.535} C_VEL
LIN {X 0,Y 227.665,Z 756.901,A -85,B 0,C 180,E1 -19905.21,E2 -19905.21} C_VEL
LIN {X 0,Y 229.042,Z 751.03,A -85,B 0,C 180,E1 -19907.971,E2 -19907.971} C_VEL
LIN {X 0,Y 231.27,Z 743.168,A -85,B 0,C 180,E1 -19910.918,E2 -19910.918} C_VEL
LIN {X 0,Y 233.629,Z 734.642,A -85,B 0,C 180,E1 -19913.487,E2 -19913.487} C_VEL
LIN {X 0,Y 236.616,Z 724.294,A -85,B 0,C 180,E1 -19915.98,E2 -19915.98} C_VEL
LIN {X 0,Y 239.283,Z 713.761,A -85,B 0,C 180,E1 -19918.027,E2 -19918.027} C_VEL
LIN {X 0,Y 242.047,Z 702.246,A -85,B 0,C 180,E1 -19919.815,E2 -19919.815} C_VEL
LIN {X 0,Y 244.777,Z 689.551,A -85,B 0,C 180,E1 -19921.356,E2 -19921.356} C_VEL
LIN {X 0,Y 247.13,Z 676.34,A -85,B 0,C 180,E1 -19922.582,E2 -19922.582} C_VEL
LIN {X 0,Y 249.043,Z 662.662,A -85,B 0,C 180,E1 -19923.505,E2 -19923.505} C_VEL
LIN {X 0,Y 250.345,Z 648.107,A -85,B 0,C 180,E1 -19924.154,E2 -19924.154} C_VEL
LIN {X 0,Y 254.012,Z 568.724,A -85,B 0,C 180,E1 -19926.426,E2 -19926.426} C_VEL
LIN {X 0,Y 252.232,Z 553.361,A -85,B 0,C 180,E1 -19927.258,E2 -19927.258} C_VEL
LIN {X 0,Y 245.033,Z 537.3,A -85,B 0,C 180,E1 -19929.072,E2 -19929.072} C_VEL
LIN {X 0,Y 238.075,Z 524.085,A -85,B 0,C 180,E1 -19930.883,E2 -19930.883} C_VEL
LIN {X 0,Y 236.392,Z 520.708,A -85,B 0,C 180,E1 -19931.389,E2 -19931.389} C_VEL
LIN {X 0,Y 233.995,Z 512.115,A -85,B 0,C 180,E1 -19935.104,E2 -19935.104} C_VEL
LIN {X 0,Y 231.546,Z 504.274,A -85,B 0,C 180,E1 -19938.845,E2 -19938.845} C_VEL
LIN {X 0,Y 228.933,Z 496.579,A -85,B 0,C 180,E1 -19942.951,E2 -19942.951} C_VEL
LIN {X 0,Y 227.912,Z 493.684,A -85,B 0,C 180,E1 -19944.677,E2 -19944.677} C_VEL
LIN {X 0,Y 227.9,Z 493.715,A -85,B 0,C 180,E1 -19949.703,E2 -19949.703} C_VEL
LIN {X 0,Y 227.915,Z 493.719,A -85,B 0,C 180,E1 -19954.424,E2 -19954.424} C_VEL
LIN {X 0,Y 227.937,Z 493.67,A -85,B 0,C 180,E1 -19958.285,E2 -19958.285} C_VEL
LIN {X 0,Y 228.024,Z 493.702,A -85,B 0,C 180,E1 -19962.825,E2 -19962.825} C_VEL
LIN {X 0,Y 228.084,Z 493.692,A -85,B 0,C 180,E1 -19967.544,E2 -19967.544} C_VEL
LIN {X 0,Y 228.315,Z 493.671,A -85,B 0,C 180,E1 -19971.147,E2 -19971.147} C_VEL
LIN {X 0,Y 228.348,Z 493.652,A -85,B 0,C 180,E1 -19972.929,E2 -19972.929} C_VEL
LIN {X 0,Y 228.546,Z 493.627,A -85,B 0,C 180,E1 -19978.238,E2 -19978.238} C_VEL
LIN {X 0,Y 228.545,Z 493.639,A -85,B 0,C 180,E1 -19981.762,E2 -19981.762} C_VEL
LIN {X 0,Y 228.345,Z 493.66,A -85,B 0,C 180,E1 -19987.072,E2 -19987.072} C_VEL
LIN {X 0,Y 228.149,Z 493.691,A -85,B 0,C 180,E1 -19990.651,E2 -19990.651} C_VEL
LIN {X 0,Y 228.055,Z 493.692,A -85,B 0,C 180,E1 -19994.273,E2 -19994.273} C_VEL
LIN {X 0,Y 227.994,Z 493.697,A -85,B 0,C 180,E1 -19997.954,E2 -19997.954} C_VEL
LIN {X 0,Y 227.921,Z 493.708,A -85,B 0,C 180,E1 -20002.331,E2 -20002.331} C_VEL
LIN {X 0,Y 227.935,Z 493.707,A -85,B 0,C 180,E1 -20006.605,E2 -20006.605} C_VEL
LIN {X 0,Y 227.902,Z 493.711,A -85,B 0,C 180,E1 -20010.298,E2 -20010.298} C_VEL
LIN {X 0,Y 227.882,Z 493.715,A -85,B 0,C 180,E1 -20013.72,E2 -20013.72} C_VEL
LIN {X 0,Y 227.864,Z 493.722,A -85,B 0,C 180,E1 -20018.088,E2 -20018.088} C_VEL
LIN {X 0,Y 227.892,Z 493.746,A -85,B 0,C 180,E1 -20018.711,E2 -20018.711} C_VEL
LIN {X 0,Y 230.416,Z 501.52,A -85,B 0,C 180,E1 -20023.336,E2 -20023.336} C_VEL
LIN {X 0,Y 233.065,Z 510.283,A -85,B 0,C 180,E1 -20027.945,E2 -20027.945} C_VEL
LIN {X 0,Y 235.087,Z 517.858,A -85,B 0,C 180,E1 -20031.526,E2 -20031.526} C_VEL
LIN {X 0,Y 244.096,Z 534.907,A -85,B 0,C 180,E1 -20033.904,E2 -20033.904} C_VEL
LIN {X 0,Y 251.229,Z 550.319,A -85,B 0,C 180,E1 -20035.665,E2 -20035.665} C_VEL
LIN {X 0,Y 253.69,Z 565.731,A -85,B 0,C 180,E1 -20036.561,E2 -20036.561} C_VEL
LIN {X 0,Y 250.846,Z 635.211,A -85,B 0,C 180,E1 -20038.372,E2 -20038.372} C_VEL
LIN {X 0,Y 249.834,Z 648.173,A -85,B 0,C 180,E1 -20038.996,E2 -20038.996} C_VEL
LIN {X 0,Y 248.192,Z 661.406,A -85,B 0,C 180,E1 -20039.946,E2 -20039.946} C_VEL
LIN {X 0,Y 246.072,Z 674.003,A -85,B 0,C 180,E1 -20041.189,E2 -20041.189} C_VEL
LIN {X 0,Y 243.562,Z 685.879,A -85,B 0,C 180,E1 -20042.74,E2 -20042.74} C_VEL
LIN {X 0,Y 240.995,Z 696.347,A -85,B 0,C 180,E1 -20044.49,E2 -20044.49} C_VEL
LIN {X 0,Y 238.451,Z 706.124,A -85,B 0,C 180,E1 -20046.556,E2 -20046.556} C_VEL
LIN {X 0,Y 235.57,Z 715.53,A -85,B 0,C 180,E1 -20049.025,E2 -20049.025} C_VEL
LIN {X 0,Y 233.135,Z 723.113,A -85,B 0,C 180,E1 -20051.549,E2 -20051.549} C_VEL
LIN {X 0,Y 231.095,Z 729.255,A -85,B 0,C 180,E1 -20054.118,E2 -20054.118} C_VEL
LIN {X 0,Y 229.33,Z 734.206,A -85,B 0,C 180,E1 -20056.715,E2 -20056.715} C_VEL
LIN {X 0,Y 228.014,Z 738.085,A -85,B 0,C 180,E1 -20059.345,E2 -20059.345} C_VEL
LIN {X 0,Y 227.112,Z 740.993,A -85,B 0,C 180,E1 -20061.993,E2 -20061.993} C_VEL
LIN {X 0,Y 226.581,Z 743.037,A -85,B 0,C 180,E1 -20064.663,E2 -20064.663} C_VEL
LIN {X 0,Y 226.076,Z 744.5,A -85,B 0,C 180,E1 -20068.221,E2 -20068.221} C_VEL
LIN {X 0,Y 226.075,Z 744.533,A -85,B 0,C 180,E1 -20071.784,E2 -20071.784} C_VEL
LIN {X 0,Y 226.569,Z 743.112,A -85,B 0,C 180,E1 -20075.342,E2 -20075.342} C_VEL
LIN {X 0,Y 227.418,Z 740.258,A -85,B 0,C 180,E1 -20078.891,E2 -20078.891} C_VEL
LIN {X 0,Y 228.387,Z 737.058,A -85,B 0,C 180,E1 -20081.54,E2 -20081.54} C_VEL
LIN {X 0,Y 229.841,Z 732.876,A -85,B 0,C 180,E1 -20084.162,E2 -20084.162} C_VEL
LIN {X 0,Y 231.962,Z 726.626,A -85,B 0,C 180,E1 -20087.184,E2 -20087.184} C_VEL
LIN {X 0,Y 234.212,Z 719.874,A -85,B 0,C 180,E1 -20089.732,E2 -20089.732} C_VEL
LIN {X 0,Y 236.937,Z 711.526,A -85,B 0,C 180,E1 -20092.224,E2 -20092.224} C_VEL
LIN {X 0,Y 239.686,Z 701.876,A -85,B 0,C 180,E1 -20094.522,E2 -20094.522} C_VEL
LIN {X 0,Y 242.241,Z 691.547,A -85,B 0,C 180,E1 -20096.494,E2 -20096.494} C_VEL
LIN {X 0,Y 244.75,Z 681.103,A -85,B 0,C 180,E1 -20098.05,E2 -20098.05} C_VEL
LIN {X 0,Y 246.969,Z 669.708,A -85,B 0,C 180,E1 -20099.401,E2 -20099.401} C_VEL
LIN {X 0,Y 248.926,Z 656.835,A -85,B 0,C 180,E1 -20100.546,E2 -20100.546} C_VEL
LIN {X 0,Y 250.289,Z 644.045,A -85,B 0,C 180,E1 -20101.358,E2 -20101.358} C_VEL
LIN {X 0,Y 251.208,Z 630.943,A -85,B 0,C 180,E1 -20101.877,E2 -20101.877} C_VEL
LIN {X 0,Y 253.639,Z 564.37,A -85,B 0,C 180,E1 -20103.626,E2 -20103.626} C_VEL
LIN {X 0,Y 251.126,Z 550.072,A -85,B 0,C 180,E1 -20104.5,E2 -20104.5} C_VEL
LIN {X 0,Y 243.583,Z 533.781,A -85,B 0,C 180,E1 -20106.373,E2 -20106.373} C_VEL
LIN {X 0,Y 236.638,Z 520.899,A -85,B 0,C 180,E1 -20108.178,E2 -20108.178} C_VEL
LIN {X 0,Y 235.085,Z 517.747,A -85,B 0,C 180,E1 -20108.68,E2 -20108.68} C_VEL
LIN {X 0,Y 232.727,Z 509.266,A -85,B 0,C 180,E1 -20112.75,E2 -20112.75} C_VEL
LIN {X 0,Y 230.247,Z 501.047,A -85,B 0,C 180,E1 -20117.105,E2 -20117.105} C_VEL
LIN {X 0,Y 227.914,Z 493.703,A -85,B 0,C 180,E1 -20121.544,E2 -20121.544} C_VEL
LIN {X 0,Y 227.966,Z 493.81,A -85,B 0,C 180,E1 -20122.562,E2 -20122.562} C_VEL
LIN {X 0,Y 231.123,Z 507.556,A -85,B 0,C 180,E1 -20126.169,E2 -20126.169} C_VEL
LIN {X 0,Y 234.73,Z 523.768,A -85,B 0,C 180,E1 -20130.263,E2 -20130.263} C_VEL
LIN {X 0,Y 235.021,Z 525.583,A -85,B 0,C 180,E1 -20130.708,E2 -20130.708} C_VEL
LIN {X 0,Y 233.948,Z 536.446,A -85,B 0,C 180,E1 -20133.096,E2 -20133.096} C_VEL
LIN {X 0,Y 235.818,Z 558.641,A -85,B 0,C 180,E1 -20134.324,E2 -20134.324} C_VEL
LIN {X 0,Y 236.541,Z 566.003,A -85,B 0,C 180,E1 -20134.73,E2 -20134.73} C_VEL
LIN {X 0,Y 232.683,Z 648.669,A -85,B 0,C 180,E1 -20138.874,E2 -20138.874} C_VEL
LIN {X 0,Y 231.92,Z 662.175,A -85,B 0,C 180,E1 -20139.867,E2 -20139.867} C_VEL
LIN {X 0,Y 230.989,Z 674.93,A -85,B 0,C 180,E1 -20141.139,E2 -20141.139} C_VEL
LIN {X 0,Y 230.031,Z 686.884,A -85,B 0,C 180,E1 -20142.669,E2 -20142.669} C_VEL
LIN {X 0,Y 229.548,Z 692.336,A -85,B 0,C 180,E1 -20143.499,E2 -20143.499} C_VEL
LIN {X 0,Y 228.449,Z 697.187,A -85,B 0,C 180,E1 -20144.313,E2 -20144.313} C_VEL
LIN {X 0,Y 224.89,Z 704.55,A -85,B 0,C 180,E1 -20145.729,E2 -20145.729} C_VEL
LIN {X 0,Y 221.356,Z 711.539,A -85,B 0,C 180,E1 -20147.307,E2 -20147.307} C_VEL
LIN {X 0,Y 220.312,Z 715.722,A -85,B 0,C 180,E1 -20148.352,E2 -20148.352} C_VEL
LIN {X 0,Y 219.634,Z 724.355,A -85,B 0,C 180,E1 -20150.793,E2 -20150.793} C_VEL
LIN {X 0,Y 219.134,Z 732.193,A -85,B 0,C 180,E1 -20153.556,E2 -20153.556} C_VEL
LIN {X 0,Y 218.905,Z 738.542,A -85,B 0,C 180,E1 -20156.318,E2 -20156.318} C_VEL
LIN {X 0,Y 218.789,Z 743.596,A -85,B 0,C 180,E1 -20159.079,E2 -20159.079} C_VEL
LIN {X 0,Y 218.932,Z 747.51,A -85,B 0,C 180,E1 -20161.839,E2 -20161.839} C_VEL
LIN {X 0,Y 219.105,Z 749.52,A -85,B 0,C 180,E1 -20163.678,E2 -20163.678} C_VEL
LIN {X 0,Y 219.864,Z 752.271,A -85,B 0,C 180,E1 -20167.346,E2 -20167.346} C_VEL
LIN {X 0,Y 220.676,Z 753.071,A -85,B 0,C 180,E1 -20169.162,E2 -20169.162} C_VEL
LIN {X 0,Y 221.604,Z 753.449,A -85,B 0,C 180,E1 -20170.969,E2 -20170.969} C_VEL
LIN {X 0,Y 224.074,Z 753.022,A -85,B 0,C 180,E1 -20174.532,E2 -20174.532} C_VEL
LIN {X 0,Y 225.587,Z 752.242,A -85,B 0,C 180,E1 -20176.283,E2 -20176.283} C_VEL
LIN {X 0,Y 227.475,Z 751.047,A -85,B 0,C 180,E1 -20177.996,E2 -20177.996} C_VEL
LIN {X 0,Y 230.594,Z 748.514,A -85,B 0,C 180,E1 -20180.517,E2 -20180.517} C_VEL
LIN {X 0,Y 235.558,Z 743.596,A -85,B 0,C 180,E1 -20183.752,E2 -20183.752} C_VEL
LIN {X 0,Y 239.785,Z 738.704,A -85,B 0,C 180,E1 -20186.081,E2 -20186.081} C_VEL
LIN {X 0,Y 245.374,Z 731.539,A -85,B 0,C 180,E1 -20188.669,E2 -20188.669} C_VEL
LIN {X 0,Y 251.496,Z 722.513,A -85,B 0,C 180,E1 -20191.13,E2 -20191.13} C_VEL
LIN {X 0,Y 257.145,Z 712.943,A -85,B 0,C 180,E1 -20193.135,E2 -20193.135} C_VEL
LIN {X 0,Y 262.712,Z 702.387,A -85,B 0,C 180,E1 -20194.877,E2 -20194.877} C_VEL
LIN {X 0,Y 268.07,Z 690.51,A -85,B 0,C 180,E1 -20196.382,E2 -20196.382} C_VEL
LIN {X 0,Y 272.605,Z 678.835,A -85,B 0,C 180,E1 -20197.522,E2 -20197.522} C_VEL
LIN {X 0,Y 276.619,Z 666.175,A -85,B 0,C 180,E1 -20198.496,E2 -20198.496} C_VEL
LIN {X 0,Y 280.106,Z 652.52,A -85,B 0,C 180,E1 -20199.253,E2 -20199.253} C_VEL
LIN {X 0,Y 292.513,Z 598.314,A -85,B 0,C 180,E1 -20201.706,E2 -20201.706} C_VEL
LIN {X 0,Y 292.444,Z 595.976,A -85,B 0,C 180,E1 -20203.169,E2 -20203.169} C_VEL
LIN {X 0,Y 292.537,Z 594.733,A -85,B 0,C 180,E1 -20204.851,E2 -20204.851} C_VEL
LIN {X 0,Y 292.87,Z 594.535,A -85,B 0,C 180,E1 -20206.185,E2 -20206.185} C_VEL
LIN {X 0,Y 275.607,Z 665.968,A -85,B 0,C 180,E1 -20209.437,E2 -20209.437} C_VEL
LIN {X 0,Y 271.738,Z 678.663,A -85,B 0,C 180,E1 -20210.198,E2 -20210.198} C_VEL
LIN {X 0,Y 266.803,Z 692.025,A -85,B 0,C 180,E1 -20211.271,E2 -20211.271} C_VEL
LIN {X 0,Y 261.482,Z 704.323,A -85,B 0,C 180,E1 -20212.545,E2 -20212.545} C_VEL
LIN {X 0,Y 255.5,Z 716.44,A -85,B 0,C 180,E1 -20214.229,E2 -20214.229} C_VEL
LIN {X 0,Y 250.443,Z 725.778,A -85,B 0,C 180,E1 -20215.856,E2 -20215.856} C_VEL
LIN {X 0,Y 244.109,Z 736.575,A -85,B 0,C 180,E1 -20218.301,E2 -20218.301} C_VEL
LIN {X 0,Y 238.22,Z 745.541,A -85,B 0,C 180,E1 -20220.868,E2 -20220.868} C_VEL
LIN {X 0,Y 233.824,Z 751.843,A -85,B 0,C 180,E1 -20223.199,E2 -20223.199} C_VEL
LIN {X 0,Y 230.007,Z 757.095,A -85,B 0,C 180,E1 -20225.636,E2 -20225.636} C_VEL
LIN {X 0,Y 225.793,Z 762.549,A -85,B 0,C 180,E1 -20229.031,E2 -20229.031} C_VEL
LIN {X 0,Y 223.359,Z 765.609,A -85,B 0,C 180,E1 -20231.658,E2 -20231.658} C_VEL
LIN {X 0,Y 220.865,Z 768.371,A -85,B 0,C 180,E1 -20235.25,E2 -20235.25} C_VEL
LIN {X 0,Y 219.358,Z 769.674,A -85,B 0,C 180,E1 -20238.915,E2 -20238.915} C_VEL
LIN {X 0,Y 218.788,Z 769.418,A -85,B 0,C 180,E1 -20242.615,E2 -20242.615} C_VEL
LIN {X 0,Y 218.798,Z 768.765,A -85,B 0,C 180,E1 -20244.597,E2 -20244.597} C_VEL
LIN {X 0,Y 218.856,Z 770.188,A -85,B 0,C 180,E1 -20248.157,E2 -20248.157} C_VEL
LIN {X 0,Y 218.902,Z 770.378,A -85,B 0,C 180,E1 -20249.998,E2 -20249.998} C_VEL
LIN {X 0,Y 218.851,Z 770.179,A -85,B 0,C 180,E1 -20251.838,E2 -20251.838} C_VEL
LIN {X 0,Y 218.741,Z 768.656,A -85,B 0,C 180,E1 -20255.529,E2 -20255.529} C_VEL
LIN {X 0,Y 218.918,Z 765.64,A -85,B 0,C 180,E1 -20259.234,E2 -20259.234} C_VEL
LIN {X 0,Y 219.641,Z 761.06,A -85,B 0,C 180,E1 -20262.941,E2 -20262.941} C_VEL
LIN {X 0,Y 220.726,Z 756.479,A -85,B 0,C 180,E1 -20265.7,E2 -20265.7} C_VEL
LIN {X 0,Y 222.168,Z 750.84,A -85,B 0,C 180,E1 -20268.439,E2 -20268.439} C_VEL
LIN {X 0,Y 224.574,Z 742.735,A -85,B 0,C 180,E1 -20271.572,E2 -20271.572} C_VEL
LIN {X 0,Y 227.07,Z 734.2,A -85,B 0,C 180,E1 -20274.208,E2 -20274.208} C_VEL
LIN {X 0,Y 230.216,Z 723.831,A -85,B 0,C 180,E1 -20276.759,E2 -20276.759} C_VEL
LIN {X 0,Y 232.994,Z 713.276,A -85,B 0,C 180,E1 -20278.854,E2 -20278.854} C_VEL
LIN {X 0,Y 235.876,Z 701.729,A -85,B 0,C 180,E1 -20280.677,E2 -20280.677} C_VEL
LIN {X 0,Y 238.711,Z 688.988,A -85,B 0,C 180,E1 -20282.248,E2 -20282.248} C_VEL
LIN {X 0,Y 241.156,Z 675.704,A -85,B 0,C 180,E1 -20283.494,E2 -20283.494} C_VEL
LIN {X 0,Y 243.121,Z 661.822,A -85,B 0,C 180,E1 -20284.434,E2 -20284.434} C_VEL
LIN {X 0,Y 244.405,Z 648.329,A -85,B 0,C 180,E1 -20285.041,E2 -20285.041} C_VEL
LIN {X 0,Y 248.186,Z 569.664,A -85,B 0,C 180,E1 -20287.334,E2 -20287.334} C_VEL
LIN {X 0,Y 246.67,Z 556.163,A -85,B 0,C 180,E1 -20288.087,E2 -20288.087} C_VEL
LIN {X 0,Y 240.728,Z 542.708,A -85,B 0,C 180,E1 -20289.654,E2 -20289.654} C_VEL
LIN {X 0,Y 233.836,Z 529.103,A -85,B 0,C 180,E1 -20291.534,E2 -20291.534} C_VEL
LIN {X 0,Y 229.214,Z 520.571,A -85,B 0,C 180,E1 -20292.932,E2 -20292.932} C_VEL
LIN {X 0,Y 226.67,Z 511.775,A -85,B 0,C 180,E1 -20296.991,E2 -20296.991} C_VEL
LIN {X 0,Y 224.061,Z 503.818,A -85,B 0,C 180,E1 -20301.147,E2 -20301.147} C_VEL
LIN {X 0,Y 222.188,Z 498.592,A -85,B 0,C 180,E1 -20304.185,E2 -20304.185} C_VEL
LIN {X 0,Y 220.82,Z 494.593,A -85,B 0,C 180,E1 -20306.725,E2 -20306.725} C_VEL
LIN {X 0,Y 220.859,Z 494.589,A -85,B 0,C 180,E1 -20309.394,E2 -20309.394} C_VEL
LIN {X 0,Y 220.885,Z 494.593,A -85,B 0,C 180,E1 -20313.548,E2 -20313.548} C_VEL
LIN {X 0,Y 220.855,Z 494.551,A -85,B 0,C 180,E1 -20317.551,E2 -20317.551} C_VEL
LIN {X 0,Y 220.974,Z 494.582,A -85,B 0,C 180,E1 -20322.571,E2 -20322.571} C_VEL
LIN {X 0,Y 221.017,Z 494.577,A -85,B 0,C 180,E1 -20327.139,E2 -20327.139} C_VEL
LIN {X 0,Y 221.248,Z 494.551,A -85,B 0,C 180,E1 -20330.861,E2 -20330.861} C_VEL
LIN {X 0,Y 221.301,Z 494.531,A -85,B 0,C 180,E1 -20332.702,E2 -20332.702} C_VEL
LIN {X 0,Y 221.504,Z 494.504,A -85,B 0,C 180,E1 -20338.182,E2 -20338.182} C_VEL
LIN {X 0,Y 221.503,Z 494.514,A -85,B 0,C 180,E1 -20341.818,E2 -20341.818} C_VEL
LIN {X 0,Y 221.28,Z 494.537,A -85,B 0,C 180,E1 -20347.299,E2 -20347.299} C_VEL
LIN {X 0,Y 221.097,Z 494.57,A -85,B 0,C 180,E1 -20350.995,E2 -20350.995} C_VEL
LIN {X 0,Y 221.007,Z 494.574,A -85,B 0,C 180,E1 -20356.631,E2 -20356.631} C_VEL
LIN {X 0,Y 220.884,Z 494.596,A -85,B 0,C 180,E1 -20360.487,E2 -20360.487} C_VEL
LIN {X 0,Y 220.859,Z 494.601,A -85,B 0,C 180,E1 -20364.436,E2 -20364.436} C_VEL
LIN {X 0,Y 220.83,Z 494.603,A -85,B 0,C 180,E1 -20368.515,E2 -20368.515} C_VEL
LIN {X 0,Y 220.817,Z 494.6,A -85,B 0,C 180,E1 -20372.756,E2 -20372.756} C_VEL
LIN {X 0,Y 220.874,Z 494.695,A -85,B 0,C 180,E1 -20376.77,E2 -20376.77} C_VEL
LIN {X 0,Y 223.201,Z 501.916,A -85,B 0,C 180,E1 -20381.394,E2 -20381.394} C_VEL
LIN {X 0,Y 225.006,Z 507.572,A -85,B 0,C 180,E1 -20384.65,E2 -20384.65} C_VEL
LIN {X 0,Y 227.144,Z 514.951,A -85,B 0,C 180,E1 -20388.535,E2 -20388.535} C_VEL
LIN {X 0,Y 228.07,Z 518.224,A -85,B 0,C 180,E1 -20390.057,E2 -20390.057} C_VEL
LIN {X 0,Y 236.055,Z 532.759,A -85,B 0,C 180,E1 -20392.298,E2 -20392.298} C_VEL
LIN {X 0,Y 243.217,Z 547.416,A -85,B 0,C 180,E1 -20394.184,E2 -20394.184} C_VEL
LIN {X 0,Y 245.83,Z 553.65,A -85,B 0,C 180,E1 -20394.86,E2 -20394.86} C_VEL
LIN {X 0,Y 247.854,Z 567.103,A -85,B 0,C 180,E1 -20395.655,E2 -20395.655} C_VEL
LIN {X 0,Y 244.867,Z 636.265,A -85,B 0,C 180,E1 -20397.506,E2 -20397.506} C_VEL
LIN {X 0,Y 243.811,Z 648.942,A -85,B 0,C 180,E1 -20398.141,E2 -20398.141} C_VEL
LIN {X 0,Y 242.097,Z 662.042,A -85,B 0,C 180,E1 -20399.108,E2 -20399.108} C_VEL
LIN {X 0,Y 239.913,Z 674.561,A -85,B 0,C 180,E1 -20400.377,E2 -20400.377} C_VEL
LIN {X 0,Y 237.288,Z 686.372,A -85,B 0,C 180,E1 -20401.956,E2 -20401.956} C_VEL
LIN {X 0,Y 234.305,Z 697.978,A -85,B 0,C 180,E1 -20403.972,E2 -20403.972} C_VEL
LIN {X 0,Y 231.45,Z 708.315,A -85,B 0,C 180,E1 -20406.278,E2 -20406.278} C_VEL
LIN {X 0,Y 228.486,Z 717.318,A -85,B 0,C 180,E1 -20408.815,E2 -20408.815} C_VEL
LIN {X 0,Y 226.059,Z 724.621,A -85,B 0,C 180,E1 -20411.42,E2 -20411.42} C_VEL
LIN {X 0,Y 223.644,Z 731.427,A -85,B 0,C 180,E1 -20414.51,E2 -20414.51} C_VEL
LIN {X 0,Y 221.91,Z 736.002,A -85,B 0,C 180,E1 -20417.194,E2 -20417.194} C_VEL
LIN {X 0,Y 220.705,Z 739.554,A -85,B 0,C 180,E1 -20419.916,E2 -20419.916} C_VEL
LIN {X 0,Y 219.881,Z 742.186,A -85,B 0,C 180,E1 -20422.657,E2 -20422.657} C_VEL
LIN {X 0,Y 219.545,Z 743.446,A -85,B 0,C 180,E1 -20424.492,E2 -20424.492} C_VEL
LIN {X 0,Y 219.008,Z 744.909,A -85,B 0,C 180,E1 -20428.163,E2 -20428.163} C_VEL
LIN {X 0,Y 219.007,Z 744.941,A -85,B 0,C 180,E1 -20431.841,E2 -20431.841} C_VEL
LIN {X 0,Y 219.533,Z 743.52,A -85,B 0,C 180,E1 -20435.514,E2 -20435.514} C_VEL
LIN {X 0,Y 220.422,Z 740.666,A -85,B 0,C 180,E1 -20439.176,E2 -20439.176} C_VEL
LIN {X 0,Y 221.454,Z 737.467,A -85,B 0,C 180,E1 -20441.907,E2 -20441.907} C_VEL
LIN {X 0,Y 222.968,Z 733.289,A -85,B 0,C 180,E1 -20444.608,E2 -20444.608} C_VEL
LIN {X 0,Y 225.211,Z 727.041,A -85,B 0,C 180,E1 -20447.716,E2 -20447.716} C_VEL
LIN {X 0,Y 227.563,Z 720.294,A -85,B 0,C 180,E1 -20450.333,E2 -20450.333} C_VEL
LIN {X 0,Y 230.405,Z 711.961,A -85,B 0,C 180,E1 -20452.889,E2 -20452.889} C_VEL
LIN {X 0,Y 232.906,Z 703.507,A -85,B 0,C 180,E1 -20454.992,E2 -20454.992} C_VEL
LIN {X 0,Y 235.628,Z 693.176,A -85,B 0,C 180,E1 -20457.058,E2 -20457.058} C_VEL
LIN {X 0,Y 238.189,Z 683.019,A -85,B 0,C 180,E1 -20458.653,E2 -20458.653} C_VEL
LIN {X 0,Y 240.501,Z 672.013,A -85,B 0,C 180,E1 -20460.031,E2 -20460.031} C_VEL
LIN {X 0,Y 242.555,Z 659.901,A -85,B 0,C 180,E1 -20461.195,E2 -20461.195} C_VEL
LIN {X 0,Y 244.109,Z 646.751,A -85,B 0,C 180,E1 -20462.124,E2 -20462.124} C_VEL
LIN {X 0,Y 245.188,Z 633.779,A -85,B 0,C 180,E1 -20462.695,E2 -20462.695} C_VEL
LIN {X 0,Y 247.89,Z 565.884,A -85,B 0,C 180,E1 -20464.517,E2 -20464.517} C_VEL
LIN {X 0,Y 245.595,Z 552.804,A -85,B 0,C 180,E1 -20465.352,E2 -20465.352} C_VEL
LIN {X 0,Y 237.948,Z 536.318,A -85,B 0,C 180,E1 -20467.345,E2 -20467.345} C_VEL
LIN {X 0,Y 230.482,Z 522.377,A -85,B 0,C 180,E1 -20469.405,E2 -20469.405} C_VEL
LIN {X 0,Y 227.943,Z 517.844,A -85,B 0,C 180,E1 -20470.202,E2 -20470.202} C_VEL
LIN {X 0,Y 225.69,Z 509.886,A -85,B 0,C 180,E1 -20474.256,E2 -20474.256} C_VEL
LIN {X 0,Y 223.892,Z 503.974,A -85,B 0,C 180,E1 -20477.554,E2 -20477.554} C_VEL
LIN {X 0,Y 221.683,Z 497.076,A -85,B 0,C 180,E1 -20481.815,E2 -20481.815} C_VEL
LIN {X 0,Y 221.245,Z 496.144,A -85,B 0,C 180,E1 -20482.529,E2 -20482.529} C_VEL
LIN {X 0,Y 224.704,Z 511.22,A -85,B 0,C 180,E1 -20486.547,E2 -20486.547} C_VEL
LIN {X 0,Y 228.009,Z 526.415,A -85,B 0,C 180,E1 -20490.45,E2 -20490.45} C_VEL
LIN {X 0,Y 226.989,Z 536.383,A -85,B 0,C 180,E1 -20492.746,E2 -20492.746} C_VEL
LIN {X 0,Y 228.577,Z 556.682,A -85,B 0,C 180,E1 -20493.902,E2 -20493.902} C_VEL
LIN {X 0,Y 229.547,Z 566.018,A -85,B 0,C 180,E1 -20494.437,E2 -20494.437} C_VEL
LIN {X 0,Y 225.57,Z 648.812,A -85,B 0,C 180,E1 -20498.765,E2 -20498.765} C_VEL
LIN {X 0,Y 224.851,Z 661.721,A -85,B 0,C 180,E1 -20499.744,E2 -20499.744} C_VEL
LIN {X 0,Y 223.828,Z 675.953,A -85,B 0,C 180,E1 -20501.225,E2 -20501.225} C_VEL
LIN {X 0,Y 222.767,Z 689.181,A -85,B 0,C 180,E1 -20503.032,E2 -20503.032} C_VEL
LIN {X 0,Y 221.654,Z 701.008,A -85,B 0,C 180,E1 -20505.071,E2 -20505.071} C_VEL
LIN {X 0,Y 220.573,Z 712.647,A -85,B 0,C 180,E1 -20507.58,E2 -20507.58} C_VEL
LIN {X 0,Y 220.312,Z 715.722,A -85,B 0,C 180,E1 -20508.352,E2 -20508.352} C_VEL
LIN {X 0,Y 219.301,Z 719.769,A -85,B 0,C 180,E1 -20509.443,E2 -20509.443} C_VEL
LIN {X 0,Y 215.969,Z 725.709,A -85,B 0,C 180,E1 -20511.343,E2 -20511.343} C_VEL
LIN {X 0,Y 212.75,Z 731.106,A -85,B 0,C 180,E1 -20513.419,E2 -20513.419} C_VEL
LIN {X 0,Y 211.933,Z 734.288,A -85,B 0,C 180,E1 -20514.757,E2 -20514.757} C_VEL
LIN {X 0,Y 211.819,Z 739.451,A -85,B 0,C 180,E1 -20517.147,E2 -20517.147} C_VEL
LIN {X 0,Y 211.732,Z 744.364,A -85,B 0,C 180,E1 -20520,E2 -20520} C_VEL
LIN {X 0,Y 211.927,Z 748.156,A -85,B 0,C 180,E1 -20522.851,E2 -20522.851} C_VEL
LIN {X 0,Y 212.318,Z 750.951,A -85,B 0,C 180,E1 -20525.699,E2 -20525.699} C_VEL
LIN {X 0,Y 213.239,Z 752.849,A -85,B 0,C 180,E1 -20528.59,E2 -20528.59} C_VEL
LIN {X 0,Y 214.657,Z 753.794,A -85,B 0,C 180,E1 -20531.329,E2 -20531.329} C_VEL
LIN {X 0,Y 217.255,Z 753.763,A -85,B 0,C 180,E1 -20534.998,E2 -20534.998} C_VEL
LIN {X 0,Y 218.847,Z 753.157,A -85,B 0,C 180,E1 -20536.799,E2 -20536.799} C_VEL
LIN {X 0,Y 222.909,Z 750.77,A -85,B 0,C 180,E1 -20540.292,E2 -20540.292} C_VEL
LIN {X 0,Y 226.632,Z 747.921,A -85,B 0,C 180,E1 -20542.807,E2 -20542.807} C_VEL
LIN {X 0,Y 230.709,Z 744.125,A -85,B 0,C 180,E1 -20545.244,E2 -20545.244} C_VEL
LIN {X 0,Y 235.338,Z 739.293,A -85,B 0,C 180,E1 -20547.573,E2 -20547.573} C_VEL
LIN {X 0,Y 241.345,Z 732.195,A -85,B 0,C 180,E1 -20550.154,E2 -20550.154} C_VEL
LIN {X 0,Y 247.85,Z 723.287,A -85,B 0,C 180,E1 -20552.599,E2 -20552.599} C_VEL
LIN {X 0,Y 253.872,Z 713.915,A -85,B 0,C 180,E1 -20554.576,E2 -20554.576} C_VEL
LIN {X 0,Y 260.285,Z 702.491,A -85,B 0,C 180,E1 -20556.443,E2 -20556.443} C_VEL
LIN {X 0,Y 265.951,Z 690.653,A -85,B 0,C 180,E1 -20557.908,E2 -20557.908} C_VEL
LIN {X 0,Y 270.708,Z 679.068,A -85,B 0,C 180,E1 -20559.018,E2 -20559.018} C_VEL
LIN {X 0,Y 275.003,Z 666.275,A -85,B 0,C 180,E1 -20559.963,E2 -20559.963} C_VEL
LIN {X 0,Y 278.622,Z 652.832,A -85,B 0,C 180,E1 -20560.684,E2 -20560.684} C_VEL
LIN {X 0,Y 290.566,Z 603.513,A -85,B 0,C 180,E1 -20562.867,E2 -20562.867} C_VEL
LIN {X 0,Y 290.632,Z 602.215,A -85,B 0,C 180,E1 -20563.992,E2 -20563.992} C_VEL
LIN {X 0,Y 290.776,Z 601.533,A -85,B 0,C 180,E1 -20565.052,E2 -20565.052} C_VEL
LIN {X 0,Y 274.645,Z 664.876,A -85,B 0,C 180,E1 -20567.91,E2 -20567.91} C_VEL
LIN {X 0,Y 270.197,Z 678.64,A -85,B 0,C 180,E1 -20568.696,E2 -20568.696} C_VEL
LIN {X 0,Y 264.981,Z 691.751,A -85,B 0,C 180,E1 -20569.72,E2 -20569.72} C_VEL
LIN {X 0,Y 258.766,Z 705.08,A -85,B 0,C 180,E1 -20571.09,E2 -20571.09} C_VEL
LIN {X 0,Y 252.436,Z 716.902,A -85,B 0,C 180,E1 -20572.73,E2 -20572.73} C_VEL
LIN {X 0,Y 246.001,Z 727.604,A -85,B 0,C 180,E1 -20574.651,E2 -20574.651} C_VEL
LIN {X 0,Y 239.308,Z 737.907,A -85,B 0,C 180,E1 -20577.089,E2 -20577.089} C_VEL
LIN {X 0,Y 233.073,Z 746.411,A -85,B 0,C 180,E1 -20579.661,E2 -20579.661} C_VEL
LIN {X 0,Y 227.652,Z 753.34,A -85,B 0,C 180,E1 -20582.412,E2 -20582.412} C_VEL
LIN {X 0,Y 223.648,Z 758.148,A -85,B 0,C 180,E1 -20584.896,E2 -20584.896} C_VEL
LIN {X 0,Y 220.265,Z 762.052,A -85,B 0,C 180,E1 -20587.485,E2 -20587.485} C_VEL
LIN {X 0,Y 216.611,Z 765.925,A -85,B 0,C 180,E1 -20591.065,E2 -20591.065} C_VEL
LIN {X 0,Y 213.971,Z 768.312,A -85,B 0,C 180,E1 -20594.763,E2 -20594.763} C_VEL
LIN {X 0,Y 212.352,Z 769.233,A -85,B 0,C 180,E1 -20598.544,E2 -20598.544} C_VEL
LIN {X 0,Y 211.748,Z 768.696,A -85,B 0,C 180,E1 -20602.368,E2 -20602.368} C_VEL
LIN {X 0,Y 211.712,Z 768.124,A -85,B 0,C 180,E1 -20604.043,E2 -20604.043} C_VEL
LIN {X 0,Y 211.709,Z 769.209,A -85,B 0,C 180,E1 -20606.191,E2 -20606.191} C_VEL
LIN {X 0,Y 211.787,Z 769.78,A -85,B 0,C 180,E1 -20608.096,E2 -20608.096} C_VEL
LIN {X 0,Y 211.83,Z 769.97,A -85,B 0,C 180,E1 -20609.998,E2 -20609.998} C_VEL
LIN {X 0,Y 211.778,Z 769.77,A -85,B 0,C 180,E1 -20611.899,E2 -20611.899} C_VEL
LIN {X 0,Y 211.647,Z 768.244,A -85,B 0,C 180,E1 -20615.715,E2 -20615.715} C_VEL
LIN {X 0,Y 211.845,Z 765.224,A -85,B 0,C 180,E1 -20619.545,E2 -20619.545} C_VEL
LIN {X 0,Y 212.673,Z 760.644,A -85,B 0,C 180,E1 -20623.372,E2 -20623.372} C_VEL
LIN {X 0,Y 213.811,Z 756.057,A -85,B 0,C 180,E1 -20626.221,E2 -20626.221} C_VEL
LIN {X 0,Y 215.403,Z 750.416,A -85,B 0,C 180,E1 -20629.04,E2 -20629.04} C_VEL
LIN {X 0,Y 217.925,Z 742.303,A -85,B 0,C 180,E1 -20632.265,E2 -20632.265} C_VEL
LIN {X 0,Y 220.569,Z 733.761,A -85,B 0,C 180,E1 -20634.97,E2 -20634.97} C_VEL
LIN {X 0,Y 223.281,Z 725.236,A -85,B 0,C 180,E1 -20637.152,E2 -20637.152} C_VEL
LIN {X 0,Y 226.43,Z 714.04,A -85,B 0,C 180,E1 -20639.503,E2 -20639.503} C_VEL
LIN {X 0,Y 229.417,Z 702.652,A -85,B 0,C 180,E1 -20641.382,E2 -20641.382} C_VEL
LIN {X 0,Y 232.339,Z 690.2,A -85,B 0,C 180,E1 -20642.986,E2 -20642.986} C_VEL
LIN {X 0,Y 234.882,Z 677.328,A -85,B 0,C 180,E1 -20644.253,E2 -20644.253} C_VEL
LIN {X 0,Y 236.907,Z 664.194,A -85,B 0,C 180,E1 -20645.211,E2 -20645.211} C_VEL
LIN {X 0,Y 238.4,Z 649.895,A -85,B 0,C 180,E1 -20645.929,E2 -20645.929} C_VEL
LIN {X 0,Y 242.438,Z 570.828,A -85,B 0,C 180,E1 -20648.274,E2 -20648.274} C_VEL
LIN {X 0,Y 241.192,Z 558.987,A -85,B 0,C 180,E1 -20648.947,E2 -20648.947} C_VEL
LIN {X 0,Y 235.381,Z 545.658,A -85,B 0,C 180,E1 -20650.562,E2 -20650.562} C_VEL
LIN {X 0,Y 227.232,Z 529.741,A -85,B 0,C 180,E1 -20652.915,E2 -20652.915} C_VEL
LIN {X 0,Y 222.027,Z 520.546,A -85,B 0,C 180,E1 -20654.558,E2 -20654.558} C_VEL
LIN {X 0,Y 219.397,Z 511.708,A -85,B 0,C 180,E1 -20658.953,E2 -20658.953} C_VEL
LIN {X 0,Y 216.962,Z 504.214,A -85,B 0,C 180,E1 -20663.183,E2 -20663.183} C_VEL
LIN {X 0,Y 214.562,Z 497.927,A -85,B 0,C 180,E1 -20667.285,E2 -20667.285} C_VEL
LIN {X 0,Y 213.809,Z 495.466,A -85,B 0,C 180,E1 -20669.018,E2 -20669.018} C_VEL
LIN {X 0,Y 213.817,Z 495.467,A -85,B 0,C 180,E1 -20672.602,E2 -20672.602} C_VEL
LIN {X 0,Y 213.809,Z 495.431,A -85,B 0,C 180,E1 -20676.973,E2 -20676.973} C_VEL
LIN {X 0,Y 213.934,Z 495.457,A -85,B 0,C 180,E1 -20682.803,E2 -20682.803} C_VEL
LIN {X 0,Y 213.971,Z 495.457,A -85,B 0,C 180,E1 -20686.708,E2 -20686.708} C_VEL
LIN {X 0,Y 214.187,Z 495.427,A -85,B 0,C 180,E1 -20690.557,E2 -20690.557} C_VEL
LIN {X 0,Y 214.238,Z 495.413,A -85,B 0,C 180,E1 -20692.46,E2 -20692.46} C_VEL
LIN {X 0,Y 214.437,Z 495.384,A -85,B 0,C 180,E1 -20698.122,E2 -20698.122} C_VEL
LIN {X 0,Y 214.545,Z 495.379,A -85,B 0,C 180,E1 -20700,E2 -20700} C_VEL
LIN {X 0,Y 214.437,Z 495.393,A -85,B 0,C 180,E1 -20701.878,E2 -20701.878} C_VEL
LIN {X 0,Y 214.218,Z 495.415,A -85,B 0,C 180,E1 -20707.541,E2 -20707.541} C_VEL
LIN {X 0,Y 214.014,Z 495.451,A -85,B 0,C 180,E1 -20711.364,E2 -20711.364} C_VEL
LIN {X 0,Y 213.925,Z 495.462,A -85,B 0,C 180,E1 -20715.238,E2 -20715.238} C_VEL
LIN {X 0,Y 213.831,Z 495.467,A -85,B 0,C 180,E1 -20719.188,E2 -20719.188} C_VEL
LIN {X 0,Y 213.839,Z 495.465,A -85,B 0,C 180,E1 -20723.228,E2 -20723.228} C_VEL
LIN {X 0,Y 213.821,Z 495.468,A -85,B 0,C 180,E1 -20727.451,E2 -20727.451} C_VEL
LIN {X 0,Y 213.772,Z 495.479,A -85,B 0,C 180,E1 -20731.737,E2 -20731.737} C_VEL
LIN {X 0,Y 213.796,Z 495.654,A -85,B 0,C 180,E1 -20734.558,E2 -20734.558} C_VEL
LIN {X 0,Y 216.135,Z 502.444,A -85,B 0,C 180,E1 -20739.351,E2 -20739.351} C_VEL
LIN {X 0,Y 217.851,Z 507.715,A -85,B 0,C 180,E1 -20742.647,E2 -20742.647} C_VEL
LIN {X 0,Y 220.244,Z 515.873,A -85,B 0,C 180,E1 -20747.217,E2 -20747.217} C_VEL
LIN {X 0,Y 220.837,Z 518.129,A -85,B 0,C 180,E1 -20748.366,E2 -20748.366} C_VEL
LIN {X 0,Y 227.123,Z 529.103,A -85,B 0,C 180,E1 -20750.283,E2 -20750.283} C_VEL
LIN {X 0,Y 234.249,Z 542.642,A -85,B 0,C 180,E1 -20752.308,E2 -20752.308} C_VEL
LIN {X 0,Y 240.346,Z 556.168,A -85,B 0,C 180,E1 -20753.967,E2 -20753.967} C_VEL
LIN {X 0,Y 242.112,Z 567.485,A -85,B 0,C 180,E1 -20754.679,E2 -20754.679} C_VEL
LIN {X 0,Y 239.038,Z 636.135,A -85,B 0,C 180,E1 -20756.549,E2 -20756.549} C_VEL
LIN {X 0,Y 237.942,Z 648.94,A -85,B 0,C 180,E1 -20757.196,E2 -20757.196} C_VEL
LIN {X 0,Y 236.26,Z 661.544,A -85,B 0,C 180,E1 -20758.132,E2 -20758.132} C_VEL
LIN {X 0,Y 234.202,Z 673.355,A -85,B 0,C 180,E1 -20759.33,E2 -20759.33} C_VEL
LIN {X 0,Y 231.473,Z 685.564,A -85,B 0,C 180,E1 -20760.938,E2 -20760.938} C_VEL
LIN {X 0,Y 228.865,Z 695.318,A -85,B 0,C 180,E1 -20762.576,E2 -20762.576} C_VEL
LIN {X 0,Y 226.082,Z 705.268,A -85,B 0,C 180,E1 -20764.698,E2 -20764.698} C_VEL
LIN {X 0,Y 222.901,Z 714.943,A -85,B 0,C 180,E1 -20767.282,E2 -20767.282} C_VEL
LIN {X 0,Y 220.099,Z 722.788,A -85,B 0,C 180,E1 -20769.927,E2 -20769.927} C_VEL
LIN {X 0,Y 217.519,Z 730.086,A -85,B 0,C 180,E1 -20773.098,E2 -20773.098} C_VEL
LIN {X 0,Y 215.563,Z 735.033,A -85,B 0,C 180,E1 -20775.849,E2 -20775.849} C_VEL
LIN {X 0,Y 214.092,Z 738.911,A -85,B 0,C 180,E1 -20778.643,E2 -20778.643} C_VEL
LIN {X 0,Y 213.001,Z 742.152,A -85,B 0,C 180,E1 -20781.835,E2 -20781.835} C_VEL
LIN {X 0,Y 212.487,Z 743.856,A -85,B 0,C 180,E1 -20784.308,E2 -20784.308} C_VEL
LIN {X 0,Y 211.941,Z 745.317,A -85,B 0,C 180,E1 -20788.102,E2 -20788.102} C_VEL
LIN {X 0,Y 211.94,Z 745.349,A -85,B 0,C 180,E1 -20791.903,E2 -20791.903} C_VEL
LIN {X 0,Y 212.477,Z 743.929,A -85,B 0,C 180,E1 -20795.697,E2 -20795.697} C_VEL
LIN {X 0,Y 213.419,Z 741.076,A -85,B 0,C 180,E1 -20799.479,E2 -20799.479} C_VEL
LIN {X 0,Y 214.519,Z 737.878,A -85,B 0,C 180,E1 -20802.298,E2 -20802.298} C_VEL
LIN {X 0,Y 216.116,Z 733.702,A -85,B 0,C 180,E1 -20805.082,E2 -20805.082} C_VEL
LIN {X 0,Y 218.478,Z 727.456,A -85,B 0,C 180,E1 -20808.281,E2 -20808.281} C_VEL
LIN {X 0,Y 220.938,Z 720.714,A -85,B 0,C 180,E1 -20810.971,E2 -20810.971} C_VEL
LIN {X 0,Y 223.893,Z 712.397,A -85,B 0,C 180,E1 -20813.594,E2 -20813.594} C_VEL
LIN {X 0,Y 226.946,Z 702.404,A -85,B 0,C 180,E1 -20816.095,E2 -20816.095} C_VEL
LIN {X 0,Y 229.663,Z 692.487,A -85,B 0,C 180,E1 -20818.069,E2 -20818.069} C_VEL
LIN {X 0,Y 232.372,Z 682.103,A -85,B 0,C 180,E1 -20819.689,E2 -20819.689} C_VEL
LIN {X 0,Y 234.75,Z 670.803,A -85,B 0,C 180,E1 -20821.096,E2 -20821.096} C_VEL
LIN {X 0,Y 236.887,Z 658.181,A -85,B 0,C 180,E1 -20822.28,E2 -20822.28} C_VEL
LIN {X 0,Y 238.345,Z 645.745,A -85,B 0,C 180,E1 -20823.124,E2 -20823.124} C_VEL
LIN {X 0,Y 239.436,Z 631.92,A -85,B 0,C 180,E1 -20823.709,E2 -20823.709} C_VEL
LIN {X 0,Y 242.123,Z 566.622,A -85,B 0,C 180,E1 -20825.49,E2 -20825.49} C_VEL
LIN {X 0,Y 240.154,Z 555.612,A -85,B 0,C 180,E1 -20826.234,E2 -20826.234} C_VEL
LIN {X 0,Y 232.976,Z 540.066,A -85,B 0,C 180,E1 -20828.196,E2 -20828.196} C_VEL
LIN {X 0,Y 226.107,Z 527.097,A -85,B 0,C 180,E1 -20830.183,E2 -20830.183} C_VEL
LIN {X 0,Y 222.261,Z 520.815,A -85,B 0,C 180,E1 -20831.339,E2 -20831.339} C_VEL
LIN {X 0,Y 220.786,Z 517.938,A -85,B 0,C 180,E1 -20831.876,E2 -20831.876} C_VEL
LIN {X 0,Y 218.503,Z 509.922,A -85,B 0,C 180,E1 -20836.248,E2 -20836.248} C_VEL
LIN {X 0,Y 216.216,Z 502.706,A -85,B 0,C 180,E1 -20840.667,E2 -20840.667} C_VEL
LIN {X 0,Y 215.717,Z 501.04,A -85,B 0,C 180,E1 -20841.755,E2 -20841.755} C_VEL
LIN {X 0,Y 214.841,Z 499.827,A -85,B 0,C 180,E1 -20842.886,E2 -20842.886} C_VEL
LIN {X 0,Y 217.83,Z 512.864,A -85,B 0,C 180,E1 -20846.415,E2 -20846.415} C_VEL
LIN {X 0,Y 220.96,Z 527.052,A -85,B 0,C 180,E1 -20850.14,E2 -20850.14} C_VEL
LIN {X 0,Y 220.026,Z 536.707,A -85,B 0,C 180,E1 -20852.406,E2 -20852.406} C_VEL
LIN {X 0,Y 221.65,Z 557.868,A -85,B 0,C 180,E1 -20853.646,E2 -20853.646} C_VEL
LIN {X 0,Y 222.551,Z 566.168,A -85,B 0,C 180,E1 -20854.139,E2 -20854.139} C_VEL
LIN {X 0,Y 218.5,Z 648.619,A -85,B 0,C 180,E1 -20858.663,E2 -20858.663} C_VEL
LIN {X 0,Y 217.741,Z 661.97,A -85,B 0,C 180,E1 -20859.704,E2 -20859.704} C_VEL
LIN {X 0,Y 216.797,Z 674.966,A -85,B 0,C 180,E1 -20861.084,E2 -20861.084} C_VEL
LIN {X 0,Y 215.811,Z 687.01,A -85,B 0,C 180,E1 -20862.712,E2 -20862.712} C_VEL
LIN {X 0,Y 214.712,Z 699.315,A -85,B 0,C 180,E1 -20864.819,E2 -20864.819} C_VEL
LIN {X 0,Y 213.668,Z 710.29,A -85,B 0,C 180,E1 -20867.172,E2 -20867.172} C_VEL
LIN {X 0,Y 212.785,Z 720.97,A -85,B 0,C 180,E1 -20870.014,E2 -20870.014} C_VEL
LIN {X 0,Y 212.179,Z 729.655,A -85,B 0,C 180,E1 -20872.912,E2 -20872.912} C_VEL
LIN {X 0,Y 211.933,Z 734.288,A -85,B 0,C 180,E1 -20874.757,E2 -20874.757} C_VEL
LIN {X 0,Y 211.159,Z 737.285,A -85,B 0,C 180,E1 -20876.119,E2 -20876.119} C_VEL
LIN {X 0,Y 208.226,Z 741.47,A -85,B 0,C 180,E1 -20878.44,E2 -20878.44} C_VEL
LIN {X 0,Y 205.838,Z 744.345,A -85,B 0,C 180,E1 -20880.402,E2 -20880.402} C_VEL
LIN {X 0,Y 204.88,Z 746.375,A -85,B 0,C 180,E1 -20881.947,E2 -20881.947} C_VEL
LIN {X 0,Y 204.832,Z 747.028,A -85,B 0,C 180,E1 -20882.471,E2 -20882.471} C_VEL
LIN {X 0,Y 205.261,Z 750.682,A -85,B 0,C 180,E1 -20885.895,E2 -20885.895} C_VEL
LIN {X 0,Y 206.684,Z 753.34,A -85,B 0,C 180,E1 -20889.789,E2 -20889.789} C_VEL
LIN {X 0,Y 207.722,Z 754.091,A -85,B 0,C 180,E1 -20891.712,E2 -20891.712} C_VEL
LIN {X 0,Y 210.437,Z 754.396,A -85,B 0,C 180,E1 -20895.496,E2 -20895.496} C_VEL
LIN {X 0,Y 212.126,Z 753.993,A -85,B 0,C 180,E1 -20897.348,E2 -20897.348} C_VEL
LIN {X 0,Y 216.375,Z 752.056,A -85,B 0,C 180,E1 -20900.933,E2 -20900.933} C_VEL
LIN {X 0,Y 221.645,Z 748.491,A -85,B 0,C 180,E1 -20904.343,E2 -20904.343} C_VEL
LIN {X 0,Y 226.088,Z 744.749,A -85,B 0,C 180,E1 -20906.791,E2 -20906.791} C_VEL
LIN {X 0,Y 231.09,Z 739.989,A -85,B 0,C 180,E1 -20909.117,E2 -20909.117} C_VEL
LIN {X 0,Y 237.493,Z 733.009,A -85,B 0,C 180,E1 -20911.686,E2 -20911.686} C_VEL
LIN {X 0,Y 243.414,Z 725.622,A -85,B 0,C 180,E1 -20913.765,E2 -20913.765} C_VEL
LIN {X 0,Y 249.722,Z 716.753,A -85,B 0,C 180,E1 -20915.73,E2 -20915.73} C_VEL
LIN {X 0,Y 256.425,Z 705.901,A -85,B 0,C 180,E1 -20917.576,E2 -20917.576} C_VEL
LIN {X 0,Y 261.976,Z 695.612,A -85,B 0,C 180,E1 -20918.936,E2 -20918.936} C_VEL
LIN {X 0,Y 267.257,Z 684.198,A -85,B 0,C 180,E1 -20920.111,E2 -20920.111} C_VEL
LIN {X 0,Y 272.262,Z 671.183,A -85,B 0,C 180,E1 -20921.156,E2 -20921.156} C_VEL
LIN {X 0,Y 276.639,Z 656.737,A -85,B 0,C 180,E1 -20921.979,E2 -20921.979} C_VEL
LIN {X 0,Y 287.762,Z 613.069,A -85,B 0,C 180,E1 -20923.894,E2 -20923.894} C_VEL
LIN {X 0,Y 287.697,Z 613.214,A -85,B 0,C 180,E1 -20924.113,E2 -20924.113} C_VEL
LIN {X 0,Y 274.088,Z 664.013,A -85,B 0,C 180,E1 -20926.375,E2 -20926.375} C_VEL
LIN {X 0,Y 269.456,Z 677.654,A -85,B 0,C 180,E1 -20927.103,E2 -20927.103} C_VEL
LIN {X 0,Y 264.107,Z 690.425,A -85,B 0,C 180,E1 -20928.039,E2 -20928.039} C_VEL
LIN {X 0,Y 257.539,Z 703.796,A -85,B 0,C 180,E1 -20929.341,E2 -20929.341} C_VEL
LIN {X 0,Y 250.758,Z 715.649,A -85,B 0,C 180,E1 -20930.903,E2 -20930.903} C_VEL
LIN {X 0,Y 243.858,Z 726.375,A -85,B 0,C 180,E1 -20932.753,E2 -20932.753} C_VEL
LIN {X 0,Y 237.617,Z 735.307,A -85,B 0,C 180,E1 -20934.775,E2 -20934.775} C_VEL
LIN {X 0,Y 230.816,Z 744.105,A -85,B 0,C 180,E1 -20937.283,E2 -20937.283} C_VEL
LIN {X 0,Y 224.674,Z 751.293,A -85,B 0,C 180,E1 -20939.965,E2 -20939.965} C_VEL
LIN {X 0,Y 218.616,Z 757.819,A -85,B 0,C 180,E1 -20943.25,E2 -20943.25} C_VEL
LIN {X 0,Y 213.749,Z 762.726,A -85,B 0,C 180,E1 -20946.759,E2 -20946.759} C_VEL
LIN {X 0,Y 209.896,Z 766.146,A -85,B 0,C 180,E1 -20950.435,E2 -20950.435} C_VEL
LIN {X 0,Y 207.098,Z 768.166,A -85,B 0,C 180,E1 -20954.245,E2 -20954.245} C_VEL
LIN {X 0,Y 205.364,Z 768.757,A -85,B 0,C 180,E1 -20958.149,E2 -20958.149} C_VEL
LIN {X 0,Y 204.726,Z 767.86,A -85,B 0,C 180,E1 -20962.105,E2 -20962.105} C_VEL
LIN {X 0,Y 204.693,Z 767.414,A -85,B 0,C 180,E1 -20963.343,E2 -20963.343} C_VEL
LIN {X 0,Y 204.618,Z 768.799,A -85,B 0,C 180,E1 -20966.059,E2 -20966.059} C_VEL
LIN {X 0,Y 204.694,Z 769.371,A -85,B 0,C 180,E1 -20968.03,E2 -20968.03} C_VEL
LIN {X 0,Y 204.761,Z 769.563,A -85,B 0,C 180,E1 -20969.997,E2 -20969.997} C_VEL
LIN {X 0,Y 204.683,Z 769.36,A -85,B 0,C 180,E1 -20971.965,E2 -20971.965} C_VEL
LIN {X 0,Y 204.564,Z 767.833,A -85,B 0,C 180,E1 -20975.913,E2 -20975.913} C_VEL
LIN {X 0,Y 204.799,Z 764.81,A -85,B 0,C 180,E1 -20979.877,E2 -20979.877} C_VEL
LIN {X 0,Y 205.726,Z 760.228,A -85,B 0,C 180,E1 -20983.833,E2 -20983.833} C_VEL
LIN {X 0,Y 206.924,Z 755.635,A -85,B 0,C 180,E1 -20986.777,E2 -20986.777} C_VEL
LIN {X 0,Y 208.66,Z 749.992,A -85,B 0,C 180,E1 -20989.68,E2 -20989.68} C_VEL
LIN {X 0,Y 211.292,Z 741.871,A -85,B 0,C 180,E1 -20993.003,E2 -20993.003} C_VEL
LIN {X 0,Y 214.107,Z 733.322,A -85,B 0,C 180,E1 -20995.778,E2 -20995.778} C_VEL
LIN {X 0,Y 216.954,Z 724.784,A -85,B 0,C 180,E1 -20998.013,E2 -20998.013} C_VEL
LIN {X 0,Y 220.218,Z 713.558,A -85,B 0,C 180,E1 -21000.422,E2 -21000.422} C_VEL
LIN {X 0,Y 223.351,Z 702.136,A -85,B 0,C 180,E1 -21002.336,E2 -21002.336} C_VEL
LIN {X 0,Y 226.404,Z 689.638,A -85,B 0,C 180,E1 -21003.966,E2 -21003.966} C_VEL
LIN {X 0,Y 228.99,Z 676.688,A -85,B 0,C 180,E1 -21005.263,E2 -21005.263} C_VEL
LIN {X 0,Y 231.207,Z 662.675,A -85,B 0,C 180,E1 -21006.281,E2 -21006.281} C_VEL
LIN {X 0,Y 232.7,Z 648.77,A -85,B 0,C 180,E1 -21006.953,E2 -21006.953} C_VEL
LIN {X 0,Y 236.707,Z 571.106,A -85,B 0,C 180,E1 -21009.303,E2 -21009.303} C_VEL
LIN {X 0,Y 235.75,Z 561.662,A -85,B 0,C 180,E1 -21009.858,E2 -21009.858} C_VEL
LIN {X 0,Y 229.281,Z 546.984,A -85,B 0,C 180,E1 -21011.751,E2 -21011.751} C_VEL
LIN {X 0,Y 222.579,Z 533.979,A -85,B 0,C 180,E1 -21013.789,E2 -21013.789} C_VEL
LIN {X 0,Y 216.788,Z 524.023,A -85,B 0,C 180,E1 -21015.651,E2 -21015.651} C_VEL
LIN {X 0,Y 214.815,Z 520.428,A -85,B 0,C 180,E1 -21016.387,E2 -21016.387} C_VEL
LIN {X 0,Y 212.687,Z 513.371,A -85,B 0,C 180,E1 -21020.151,E2 -21020.151} C_VEL
LIN {X 0,Y 210.555,Z 506.901,A -85,B 0,C 180,E1 -21024.008,E2 -21024.008} C_VEL
LIN {X 0,Y 208.095,Z 500.432,A -85,B 0,C 180,E1 -21028.482,E2 -21028.482} C_VEL
LIN {X 0,Y 206.73,Z 496.35,A -85,B 0,C 180,E1 -21031.668,E2 -21031.668} C_VEL
LIN {X 0,Y 206.744,Z 496.314,A -85,B 0,C 180,E1 -21036.603,E2 -21036.603} C_VEL
LIN {X 0,Y 206.863,Z 496.343,A -85,B 0,C 180,E1 -21042.196,E2 -21042.196} C_VEL
LIN {X 0,Y 206.904,Z 496.337,A -85,B 0,C 180,E1 -21046.245,E2 -21046.245} C_VEL
LIN {X 0,Y 207.123,Z 496.304,A -85,B 0,C 180,E1 -21050.232,E2 -21050.232} C_VEL
LIN {X 0,Y 207.179,Z 496.294,A -85,B 0,C 180,E1 -21052.202,E2 -21052.202} C_VEL
LIN {X 0,Y 207.374,Z 496.264,A -85,B 0,C 180,E1 -21058.058,E2 -21058.058} C_VEL
LIN {X 0,Y 207.509,Z 496.255,A -85,B 0,C 180,E1 -21060,E2 -21060} C_VEL
LIN {X 0,Y 207.077,Z 496.299,A -85,B 0,C 180,E1 -21063.892,E2 -21063.892} C_VEL
LIN {X 0,Y 207.158,Z 496.292,A -85,B 0,C 180,E1 -21067.8,E2 -21067.8} C_VEL
LIN {X 0,Y 206.934,Z 496.328,A -85,B 0,C 180,E1 -21071.758,E2 -21071.758} C_VEL
LIN {X 0,Y 206.859,Z 496.344,A -85,B 0,C 180,E1 -21075.772,E2 -21075.772} C_VEL
LIN {X 0,Y 206.775,Z 496.353,A -85,B 0,C 180,E1 -21079.87,E2 -21079.87} C_VEL
LIN {X 0,Y 206.755,Z 496.356,A -85,B 0,C 180,E1 -21084.074,E2 -21084.074} C_VEL
LIN {X 0,Y 206.736,Z 496.359,A -85,B 0,C 180,E1 -21088.42,E2 -21088.42} C_VEL
LIN {X 0,Y 206.737,Z 496.481,A -85,B 0,C 180,E1 -21091.957,E2 -21091.957} C_VEL
LIN {X 0,Y 209.102,Z 503.238,A -85,B 0,C 180,E1 -21097.228,E2 -21097.228} C_VEL
LIN {X 0,Y 211.283,Z 509.916,A -85,B 0,C 180,E1 -21101.703,E2 -21101.703} C_VEL
LIN {X 0,Y 213.801,Z 518.382,A -85,B 0,C 180,E1 -21106.574,E2 -21106.574} C_VEL
LIN {X 0,Y 221.917,Z 532.016,A -85,B 0,C 180,E1 -21109.21,E2 -21109.21} C_VEL
LIN {X 0,Y 229.645,Z 547.139,A -85,B 0,C 180,E1 -21111.536,E2 -21111.536} C_VEL
LIN {X 0,Y 234.983,Z 559.13,A -85,B 0,C 180,E1 -21113.061,E2 -21113.061} C_VEL
LIN {X 0,Y 236.4,Z 569.061,A -85,B 0,C 180,E1 -21113.691,E2 -21113.691} C_VEL
LIN {X 0,Y 233.277,Z 635.996,A -85,B 0,C 180,E1 -21115.543,E2 -21115.543} C_VEL
LIN {X 0,Y 232.202,Z 648.172,A -85,B 0,C 180,E1 -21116.148,E2 -21116.148} C_VEL
LIN {X 0,Y 230.487,Z 661.047,A -85,B 0,C 180,E1 -21117.106,E2 -21117.106} C_VEL
LIN {X 0,Y 228.517,Z 672.153,A -85,B 0,C 180,E1 -21118.222,E2 -21118.222} C_VEL
LIN {X 0,Y 225.984,Z 683.258,A -85,B 0,C 180,E1 -21119.647,E2 -21119.647} C_VEL
LIN {X 0,Y 222.947,Z 694.642,A -85,B 0,C 180,E1 -21121.527,E2 -21121.527} C_VEL
LIN {X 0,Y 220.238,Z 703.884,A -85,B 0,C 180,E1 -21123.467,E2 -21123.467} C_VEL
LIN {X 0,Y 217.431,Z 712.402,A -85,B 0,C 180,E1 -21125.665,E2 -21125.665} C_VEL
LIN {X 0,Y 214.421,Z 720.803,A -85,B 0,C 180,E1 -21128.365,E2 -21128.365} C_VEL
LIN {X 0,Y 211.835,Z 727.601,A -85,B 0,C 180,E1 -21131.13,E2 -21131.13} C_VEL
LIN {X 0,Y 209.314,Z 733.896,A -85,B 0,C 180,E1 -21134.421,E2 -21134.421} C_VEL
LIN {X 0,Y 207.608,Z 738.122,A -85,B 0,C 180,E1 -21137.291,E2 -21137.291} C_VEL
LIN {X 0,Y 206.41,Z 741.371,A -85,B 0,C 180,E1 -21140.201,E2 -21140.201} C_VEL
LIN {X 0,Y 205.433,Z 744.265,A -85,B 0,C 180,E1 -21144.112,E2 -21144.112} C_VEL
LIN {X 0,Y 204.877,Z 745.725,A -85,B 0,C 180,E1 -21148.037,E2 -21148.037} C_VEL
LIN {X 0,Y 204.876,Z 745.756,A -85,B 0,C 180,E1 -21151.968,E2 -21151.968} C_VEL
LIN {X 0,Y 205.425,Z 744.338,A -85,B 0,C 180,E1 -21155.893,E2 -21155.893} C_VEL
LIN {X 0,Y 206.413,Z 741.485,A -85,B 0,C 180,E1 -21159.804,E2 -21159.804} C_VEL
LIN {X 0,Y 207.609,Z 738.287,A -85,B 0,C 180,E1 -21162.714,E2 -21162.714} C_VEL
LIN {X 0,Y 209.284,Z 734.114,A -85,B 0,C 180,E1 -21165.586,E2 -21165.586} C_VEL
LIN {X 0,Y 211.767,Z 727.871,A -85,B 0,C 180,E1 -21168.882,E2 -21168.882} C_VEL
LIN {X 0,Y 214.337,Z 721.135,A -85,B 0,C 180,E1 -21171.649,E2 -21171.649} C_VEL
LIN {X 0,Y 217.411,Z 712.833,A -85,B 0,C 180,E1 -21174.343,E2 -21174.343} C_VEL
LIN {X 0,Y 220.531,Z 703.155,A -85,B 0,C 180,E1 -21176.833,E2 -21176.833} C_VEL
LIN {X 0,Y 223.451,Z 692.957,A -85,B 0,C 180,E1 -21178.922,E2 -21178.922} C_VEL
LIN {X 0,Y 226.592,Z 681.19,A -85,B 0,C 180,E1 -21180.784,E2 -21180.784} C_VEL
LIN {X 0,Y 229.099,Z 669.513,A -85,B 0,C 180,E1 -21182.211,E2 -21182.211} C_VEL
LIN {X 0,Y 231.078,Z 657.553,A -85,B 0,C 180,E1 -21183.325,E2 -21183.325} C_VEL
LIN {X 0,Y 232.663,Z 644.735,A -85,B 0,C 180,E1 -21184.173,E2 -21184.173} C_VEL
LIN {X 0,Y 233.689,Z 631.63,A -85,B 0,C 180,E1 -21184.72,E2 -21184.72} C_VEL
LIN {X 0,Y 236.501,Z 568.2,A -85,B 0,C 180,E1 -21186.467,E2 -21186.467} C_VEL
LIN {X 0,Y 234.844,Z 558.66,A -85,B 0,C 180,E1 -21187.132,E2 -21187.132} C_VEL
LIN {X 0,Y 228.435,Z 544.533,A -85,B 0,C 180,E1 -21188.977,E2 -21188.977} C_VEL
LIN {X 0,Y 221.751,Z 531.748,A -85,B 0,C 180,E1 -21191.001,E2 -21191.001} C_VEL
LIN {X 0,Y 216.124,Z 522.35,A -85,B 0,C 180,E1 -21192.802,E2 -21192.802} C_VEL
LIN {X 0,Y 213.649,Z 518.056,A -85,B 0,C 180,E1 -21193.696,E2 -21193.696} C_VEL
LIN {X 0,Y 211.368,Z 510.191,A -85,B 0,C 180,E1 -21198.317,E2 -21198.317} C_VEL
LIN {X 0,Y 209.621,Z 504.689,A -85,B 0,C 180,E1 -21201.94,E2 -21201.94} C_VEL
LIN {X 0,Y 208.417,Z 503.391,A -85,B 0,C 180,E1 -21203.22,E2 -21203.22} C_VEL
LIN {X 0,Y 211.43,Z 516.876,A -85,B 0,C 180,E1 -21206.935,E2 -21206.935} C_VEL
LIN {X 0,Y 213.969,Z 528.564,A -85,B 0,C 180,E1 -21210.045,E2 -21210.045} C_VEL
LIN {X 0,Y 213.045,Z 536.915,A -85,B 0,C 180,E1 -21212.06,E2 -21212.06} C_VEL
LIN {X 0,Y 214.703,Z 558.983,A -85,B 0,C 180,E1 -21213.418,E2 -21213.418} C_VEL
LIN {X 0,Y 215.443,Z 567.453,A -85,B 0,C 180,E1 -21213.936,E2 -21213.936} C_VEL
LIN {X 0,Y 211.354,Z 649.34,A -85,B 0,C 180,E1 -21218.617,E2 -21218.617} C_VEL
LIN {X 0,Y 210.63,Z 662.305,A -85,B 0,C 180,E1 -21219.669,E2 -21219.669} C_VEL
LIN {X 0,Y 209.615,Z 675.786,A -85,B 0,C 180,E1 -21221.173,E2 -21221.173} C_VEL
LIN {X 0,Y 208.653,Z 687.618,A -85,B 0,C 180,E1 -21222.859,E2 -21222.859} C_VEL
LIN {X 0,Y 207.416,Z 700.975,A -85,B 0,C 180,E1 -21225.278,E2 -21225.278} C_VEL
LIN {X 0,Y 206.411,Z 711.658,A -85,B 0,C 180,E1 -21227.713,E2 -21227.713} C_VEL
LIN {X 0,Y 205.727,Z 720.564,A -85,B 0,C 180,E1 -21230.165,E2 -21230.165} C_VEL
LIN {X 0,Y 205.192,Z 728.126,A -85,B 0,C 180,E1 -21232.67,E2 -21232.67} C_VEL
LIN {X 0,Y 204.84,Z 735.239,A -85,B 0,C 180,E1 -21235.565,E2 -21235.565} C_VEL
LIN {X 0,Y 204.722,Z 740.225,A -85,B 0,C 180,E1 -21238.032,E2 -21238.032} C_VEL
LIN {X 0,Y 204.707,Z 745.042,A -85,B 0,C 180,E1 -21240.983,E2 -21240.983} C_VEL
LIN {X 0,Y 204.832,Z 747.028,A -85,B 0,C 180,E1 -21242.471,E2 -21242.471} C_VEL
LIN {X 0,Y 204.328,Z 748.84,A -85,B 0,C 180,E1 -21244.039,E2 -21244.039} C_VEL
LIN {X 0,Y 201.992,Z 751.198,A -85,B 0,C 180,E1 -21246.673,E2 -21246.673} C_VEL
LIN {X 0,Y 200.283,Z 752.629,A -85,B 0,C 180,E1 -21248.851,E2 -21248.851} C_VEL
LIN {X 0,Y 199.982,Z 753.54,A -85,B 0,C 180,E1 -21250.527,E2 -21250.527} C_VEL
LIN {X 0,Y 200.184,Z 753.771,A -85,B 0,C 180,E1 -21251.085,E2 -21251.085} C_VEL
LIN {X 0,Y 202.096,Z 754.795,A -85,B 0,C 180,E1 -21254.089,E2 -21254.089} C_VEL
LIN {X 0,Y 205.427,Z 754.781,A -85,B 0,C 180,E1 -21257.933,E2 -21257.933} C_VEL
LIN {X 0,Y 209.86,Z 753.219,A -85,B 0,C 180,E1 -21261.615,E2 -21261.615} C_VEL
LIN {X 0,Y 215.369,Z 750.16,A -85,B 0,C 180,E1 -21265.101,E2 -21265.101} C_VEL
LIN {X 0,Y 220.018,Z 746.819,A -85,B 0,C 180,E1 -21267.592,E2 -21267.592} C_VEL
LIN {X 0,Y 225.226,Z 742.458,A -85,B 0,C 180,E1 -21269.951,E2 -21269.951} C_VEL
LIN {X 0,Y 231.906,Z 736.056,A -85,B 0,C 180,E1 -21272.542,E2 -21272.542} C_VEL
LIN {X 0,Y 239.107,Z 728.043,A -85,B 0,C 180,E1 -21274.97,E2 -21274.97} C_VEL
LIN {X 0,Y 245.691,Z 719.633,A -85,B 0,C 180,E1 -21276.92,E2 -21276.92} C_VEL
LIN {X 0,Y 252.698,Z 709.399,A -85,B 0,C 180,E1 -21278.738,E2 -21278.738} C_VEL
LIN {X 0,Y 258.207,Z 700.274,A -85,B 0,C 180,E1 -21280.018,E2 -21280.018} C_VEL
LIN {X 0,Y 263.888,Z 689.266,A -85,B 0,C 180,E1 -21281.235,E2 -21281.235} C_VEL
LIN {X 0,Y 269.164,Z 677.396,A -85,B 0,C 180,E1 -21282.254,E2 -21282.254} C_VEL
LIN {X 0,Y 273.849,Z 664.188,A -85,B 0,C 180,E1 -21283.102,E2 -21283.102} C_VEL
LIN {X 0,Y 279.012,Z 645.583,A -85,B 0,C 180,E1 -21283.967,E2 -21283.967} C_VEL
LIN {X 0,Y 278.99,Z 645.633,A -85,B 0,C 180,E1 -21284.039,E2 -21284.039} C_VEL
LIN {X 0,Y 272.725,Z 667.111,A -85,B 0,C 180,E1 -21285.002,E2 -21285.002} C_VEL
LIN {X 0,Y 268.079,Z 679.477,A -85,B 0,C 180,E1 -21285.668,E2 -21285.668} C_VEL
LIN {X 0,Y 261.361,Z 694.042,A -85,B 0,C 180,E1 -21286.76,E2 -21286.76} C_VEL
LIN {X 0,Y 254.089,Z 707.256,A -85,B 0,C 180,E1 -21288.113,E2 -21288.113} C_VEL
LIN {X 0,Y 246.992,Z 718.446,A -85,B 0,C 180,E1 -21289.657,E2 -21289.657} C_VEL
LIN {X 0,Y 239.797,Z 728.56,A -85,B 0,C 180,E1 -21291.477,E2 -21291.477} C_VEL
LIN {X 0,Y 233.228,Z 736.966,A -85,B 0,C 180,E1 -21293.475,E2 -21293.475} C_VEL
LIN {X 0,Y 226.084,Z 745.236,A -85,B 0,C 180,E1 -21295.973,E2 -21295.973} C_VEL
LIN {X 0,Y 220.439,Z 751.188,A -85,B 0,C 180,E1 -21298.259,E2 -21298.259} C_VEL
LIN {X 0,Y 213.881,Z 757.571,A -85,B 0,C 180,E1 -21301.543,E2 -21301.543} C_VEL
LIN {X 0,Y 208.449,Z 762.341,A -85,B 0,C 180,E1 -21305.072,E2 -21305.072} C_VEL
LIN {X 0,Y 205.067,Z 765.002,A -85,B 0,C 180,E1 -21307.85,E2 -21307.85} C_VEL
LIN {X 0,Y 201.592,Z 767.294,A -85,B 0,C 180,E1 -21311.711,E2 -21311.711} C_VEL
LIN {X 0,Y 199.134,Z 768.206,A -85,B 0,C 180,E1 -21315.694,E2 -21315.694} C_VEL
LIN {X 0,Y 197.945,Z 767.741,A -85,B 0,C 180,E1 -21319.772,E2 -21319.772} C_VEL
LIN {X 0,Y 197.672,Z 766.702,A -85,B 0,C 180,E1 -21322.592,E2 -21322.592} C_VEL
LIN {X 0,Y 197.532,Z 768.389,A -85,B 0,C 180,E1 -21325.917,E2 -21325.917} C_VEL
LIN {X 0,Y 197.604,Z 768.961,A -85,B 0,C 180,E1 -21327.959,E2 -21327.959} C_VEL
LIN {X 0,Y 197.692,Z 769.155,A -85,B 0,C 180,E1 -21329.997,E2 -21329.997} C_VEL
LIN {X 0,Y 197.591,Z 768.95,A -85,B 0,C 180,E1 -21332.036,E2 -21332.036} C_VEL
LIN {X 0,Y 197.484,Z 767.421,A -85,B 0,C 180,E1 -21336.126,E2 -21336.126} C_VEL
LIN {X 0,Y 197.746,Z 764.394,A -85,B 0,C 180,E1 -21340.233,E2 -21340.233} C_VEL
LIN {X 0,Y 198.791,Z 759.812,A -85,B 0,C 180,E1 -21344.325,E2 -21344.325} C_VEL
LIN {X 0,Y 200.056,Z 755.214,A -85,B 0,C 180,E1 -21347.371,E2 -21347.371} C_VEL
LIN {X 0,Y 202.299,Z 748.531,A -85,B 0,C 180,E1 -21350.857,E2 -21350.857} C_VEL
LIN {X 0,Y 205.158,Z 740.134,A -85,B 0,C 180,E1 -21354.27,E2 -21354.27} C_VEL
LIN {X 0,Y 208.269,Z 731.271,A -85,B 0,C 180,E1 -21357.098,E2 -21357.098} C_VEL
LIN {X 0,Y 211.255,Z 722.442,A -85,B 0,C 180,E1 -21359.384,E2 -21359.384} C_VEL
LIN {X 0,Y 214.451,Z 711.822,A -85,B 0,C 180,E1 -21361.621,E2 -21361.621} C_VEL
LIN {X 0,Y 217.758,Z 700.185,A -85,B 0,C 180,E1 -21363.549,E2 -21363.549} C_VEL
LIN {X 0,Y 220.923,Z 687.301,A -85,B 0,C 180,E1 -21365.208,E2 -21365.208} C_VEL
LIN {X 0,Y 223.649,Z 673.763,A -85,B 0,C 180,E1 -21366.516,E2 -21366.516} C_VEL
LIN {X 0,Y 225.745,Z 660.161,A -85,B 0,C 180,E1 -21367.446,E2 -21367.446} C_VEL
LIN {X 0,Y 227.118,Z 646.075,A -85,B 0,C 180,E1 -21368.09,E2 -21368.09} C_VEL
LIN {X 0,Y 231.106,Z 572.109,A -85,B 0,C 180,E1 -21370.346,E2 -21370.346} C_VEL
LIN {X 0,Y 230.366,Z 564.439,A -85,B 0,C 180,E1 -21370.808,E2 -21370.808} C_VEL
LIN {X 0,Y 224.23,Z 550.39,A -85,B 0,C 180,E1 -21372.702,E2 -21372.702} C_VEL
LIN {X 0,Y 217.645,Z 537.536,A -85,B 0,C 180,E1 -21374.815,E2 -21374.815} C_VEL
LIN {X 0,Y 212.215,Z 528.177,A -85,B 0,C 180,E1 -21376.657,E2 -21376.657} C_VEL
LIN {X 0,Y 209.83,Z 524.257,A -85,B 0,C 180,E1 -21377.505,E2 -21377.505} C_VEL
LIN {X 0,Y 207.628,Z 520.411,A -85,B 0,C 180,E1 -21378.368,E2 -21378.368} C_VEL
LIN {X 0,Y 205.326,Z 512.998,A -85,B 0,C 180,E1 -21382.68,E2 -21382.68} C_VEL
LIN {X 0,Y 203.08,Z 506.509,A -85,B 0,C 180,E1 -21387.039,E2 -21387.039} C_VEL
LIN {X 0,Y 201.829,Z 502.99,A -85,B 0,C 180,E1 -21389.675,E2 -21389.675} C_VEL
LIN {X 0,Y 200.264,Z 499.267,A -85,B 0,C 180,E1 -21392.857,E2 -21392.857} C_VEL
LIN {X 0,Y 199.662,Z 497.227,A -85,B 0,C 180,E1 -21394.736,E2 -21394.736} C_VEL
LIN {X 0,Y 199.704,Z 497.185,A -85,B 0,C 180,E1 -21397.225,E2 -21397.225} C_VEL
LIN {X 0,Y 199.786,Z 497.224,A -85,B 0,C 180,E1 -21401.758,E2 -21401.758} C_VEL
LIN {X 0,Y 199.838,Z 497.212,A -85,B 0,C 180,E1 -21405.749,E2 -21405.749} C_VEL
LIN {X 0,Y 200.066,Z 497.179,A -85,B 0,C 180,E1 -21409.884,E2 -21409.884} C_VEL
LIN {X 0,Y 200.032,Z 497.177,A -85,B 0,C 180,E1 -21413.95,E2 -21413.95} C_VEL
LIN {X 0,Y 200.314,Z 497.143,A -85,B 0,C 180,E1 -21417.99,E2 -21417.99} C_VEL
LIN {X 0,Y 200.473,Z 497.13,A -85,B 0,C 180,E1 -21420,E2 -21420} C_VEL
LIN {X 0,Y 200.022,Z 497.178,A -85,B 0,C 180,E1 -21424.03,E2 -21424.03} C_VEL
LIN {X 0,Y 200.102,Z 497.169,A -85,B 0,C 180,E1 -21428.076,E2 -21428.076} C_VEL
LIN {X 0,Y 199.877,Z 497.202,A -85,B 0,C 180,E1 -21432.18,E2 -21432.18} C_VEL
LIN {X 0,Y 199.796,Z 497.218,A -85,B 0,C 180,E1 -21436.345,E2 -21436.345} C_VEL
LIN {X 0,Y 199.691,Z 497.234,A -85,B 0,C 180,E1 -21440.607,E2 -21440.607} C_VEL
LIN {X 0,Y 199.664,Z 497.235,A -85,B 0,C 180,E1 -21444.986,E2 -21444.986} C_VEL
LIN {X 0,Y 199.662,Z 497.236,A -85,B 0,C 180,E1 -21448.858,E2 -21448.858} C_VEL
LIN {X 0,Y 200.779,Z 500.239,A -85,B 0,C 180,E1 -21451.672,E2 -21451.672} C_VEL
LIN {X 0,Y 202.659,Z 505.689,A -85,B 0,C 180,E1 -21456.125,E2 -21456.125} C_VEL
LIN {X 0,Y 204.746,Z 512.184,A -85,B 0,C 180,E1 -21460.707,E2 -21460.707} C_VEL
LIN {X 0,Y 206.608,Z 518.429,A -85,B 0,C 180,E1 -21464.543,E2 -21464.543} C_VEL
LIN {X 0,Y 209.448,Z 522.943,A -85,B 0,C 180,E1 -21465.584,E2 -21465.584} C_VEL
LIN {X 0,Y 215.88,Z 533.647,A -85,B 0,C 180,E1 -21467.799,E2 -21467.799} C_VEL
LIN {X 0,Y 222.68,Z 546.538,A -85,B 0,C 180,E1 -21469.987,E2 -21469.987} C_VEL
LIN {X 0,Y 229.139,Z 560.619,A -85,B 0,C 180,E1 -21471.944,E2 -21471.944} C_VEL
LIN {X 0,Y 229.83,Z 563.034,A -85,B 0,C 180,E1 -21472.177,E2 -21472.177} C_VEL
LIN {X 0,Y 230.804,Z 570.147,A -85,B 0,C 180,E1 -21472.642,E2 -21472.642} C_VEL
LIN {X 0,Y 227.502,Z 637.041,A -85,B 0,C 180,E1 -21474.539,E2 -21474.539} C_VEL
LIN {X 0,Y 226.298,Z 649.703,A -85,B 0,C 180,E1 -21475.207,E2 -21475.207} C_VEL
LIN {X 0,Y 224.389,Z 662.812,A -85,B 0,C 180,E1 -21476.228,E2 -21476.228} C_VEL
LIN {X 0,Y 222.18,Z 674.469,A -85,B 0,C 180,E1 -21477.473,E2 -21477.473} C_VEL
LIN {X 0,Y 219.233,Z 686.56,A -85,B 0,C 180,E1 -21479.145,E2 -21479.145} C_VEL
LIN {X 0,Y 216.036,Z 697.423,A -85,B 0,C 180,E1 -21481.089,E2 -21481.089} C_VEL
LIN {X 0,Y 213.32,Z 706.301,A -85,B 0,C 180,E1 -21483.109,E2 -21483.109} C_VEL
LIN {X 0,Y 209.922,Z 715.811,A -85,B 0,C 180,E1 -21485.791,E2 -21485.791} C_VEL
LIN {X 0,Y 206.832,Z 723.641,A -85,B 0,C 180,E1 -21488.578,E2 -21488.578} C_VEL
LIN {X 0,Y 203.992,Z 730.918,A -85,B 0,C 180,E1 -21491.939,E2 -21491.939} C_VEL
LIN {X 0,Y 201.857,Z 735.859,A -85,B 0,C 180,E1 -21494.866,E2 -21494.866} C_VEL
LIN {X 0,Y 200.199,Z 739.737,A -85,B 0,C 180,E1 -21497.844,E2 -21497.844} C_VEL
LIN {X 0,Y 198.833,Z 743.345,A -85,B 0,C 180,E1 -21501.771,E2 -21501.771} C_VEL
LIN {X 0,Y 198.063,Z 745.578,A -85,B 0,C 180,E1 -21505.933,E2 -21505.933} C_VEL
LIN {X 0,Y 197.744,Z 746.336,A -85,B 0,C 180,E1 -21510.003,E2 -21510.003} C_VEL
LIN {X 0,Y 198.058,Z 745.629,A -85,B 0,C 180,E1 -21514.072,E2 -21514.072} C_VEL
LIN {X 0,Y 198.824,Z 743.505,A -85,B 0,C 180,E1 -21518.131,E2 -21518.131} C_VEL
LIN {X 0,Y 200.201,Z 739.892,A -85,B 0,C 180,E1 -21522.162,E2 -21522.162} C_VEL
LIN {X 0,Y 201.835,Z 736.048,A -85,B 0,C 180,E1 -21525.141,E2 -21525.141} C_VEL
LIN {X 0,Y 203.893,Z 731.16,A -85,B 0,C 180,E1 -21528.075,E2 -21528.075} C_VEL
LIN {X 0,Y 206.784,Z 723.964,A -85,B 0,C 180,E1 -21531.432,E2 -21531.432} C_VEL
LIN {X 0,Y 209.883,Z 716.202,A -85,B 0,C 180,E1 -21534.22,E2 -21534.22} C_VEL
LIN {X 0,Y 213.318,Z 706.49,A -85,B 0,C 180,E1 -21536.983,E2 -21536.983} C_VEL
LIN {X 0,Y 216.321,Z 696.829,A -85,B 0,C 180,E1 -21539.168,E2 -21539.168} C_VEL
LIN {X 0,Y 219.474,Z 685.931,A -85,B 0,C 180,E1 -21541.09,E2 -21541.09} C_VEL
LIN {X 0,Y 222.405,Z 673.651,A -85,B 0,C 180,E1 -21542.764,E2 -21542.764} C_VEL
LIN {X 0,Y 224.895,Z 660.629,A -85,B 0,C 180,E1 -21544.096,E2 -21544.096} C_VEL
LIN {X 0,Y 226.535,Z 648.277,A -85,B 0,C 180,E1 -21545.028,E2 -21545.028} C_VEL
LIN {X 0,Y 227.766,Z 635.966,A -85,B 0,C 180,E1 -21545.623,E2 -21545.623} C_VEL
LIN {X 0,Y 230.885,Z 568.94,A -85,B 0,C 180,E1 -21547.536,E2 -21547.536} C_VEL
LIN {X 0,Y 229.606,Z 561.645,A -85,B 0,C 180,E1 -21548.072,E2 -21548.072} C_VEL
LIN {X 0,Y 222.806,Z 546.723,A -85,B 0,C 180,E1 -21550.137,E2 -21550.137} C_VEL
LIN {X 0,Y 217.092,Z 535.812,A -85,B 0,C 180,E1 -21551.964,E2 -21551.964} C_VEL
LIN {X 0,Y 211.911,Z 527.013,A -85,B 0,C 180,E1 -21553.713,E2 -21553.713} C_VEL
LIN {X 0,Y 208.759,Z 522.027,A -85,B 0,C 180,E1 -21554.831,E2 -21554.831} C_VEL
LIN {X 0,Y 206.478,Z 518.131,A -85,B 0,C 180,E1 -21555.738,E2 -21555.738} C_VEL
LIN {X 0,Y 204.841,Z 512.445,A -85,B 0,C 180,E1 -21559.316,E2 -21559.316} C_VEL
LIN {X 0,Y 203.789,Z 509.052,A -85,B 0,C 180,E1 -21561.628,E2 -21561.628} C_VEL
LIN {X 0,Y 202.01,Z 507.003,A -85,B 0,C 180,E1 -21563.615,E2 -21563.615} C_VEL
LIN {X 0,Y 205.537,Z 523.065,A -85,B 0,C 180,E1 -21568.074,E2 -21568.074} C_VEL
LIN {X 0,Y 206.926,Z 529.941,A -85,B 0,C 180,E1 -21569.936,E2 -21569.936} C_VEL
LIN {X 0,Y 206.068,Z 537.538,A -85,B 0,C 180,E1 -21571.746,E2 -21571.746} C_VEL
LIN {X 0,Y 207.645,Z 559.115,A -85,B 0,C 180,E1 -21573.116,E2 -21573.116} C_VEL
LIN {X 0,Y 208.426,Z 567.411,A -85,B 0,C 180,E1 -21573.645,E2 -21573.645} C_VEL
LIN {X 0,Y 204.348,Z 648.339,A -85,B 0,C 180,E1 -21578.49,E2 -21578.49} C_VEL
LIN {X 0,Y 203.556,Z 661.793,A -85,B 0,C 180,E1 -21579.613,E2 -21579.613} C_VEL
LIN {X 0,Y 202.628,Z 674.345,A -85,B 0,C 180,E1 -21581.024,E2 -21581.024} C_VEL
LIN {X 0,Y 201.512,Z 688.048,A -85,B 0,C 180,E1 -21583.017,E2 -21583.017} C_VEL
LIN {X 0,Y 200.223,Z 701.367,A -85,B 0,C 180,E1 -21585.517,E2 -21585.517} C_VEL
LIN {X 0,Y 199.193,Z 713.047,A -85,B 0,C 180,E1 -21588.295,E2 -21588.295} C_VEL
LIN {X 0,Y 198.529,Z 721.704,A -85,B 0,C 180,E1 -21590.833,E2 -21590.833} C_VEL
LIN {X 0,Y 197.963,Z 730.18,A -85,B 0,C 180,E1 -21593.886,E2 -21593.886} C_VEL
LIN {X 0,Y 197.745,Z 737.104,A -85,B 0,C 180,E1 -21596.944,E2 -21596.944} C_VEL
LIN {X 0,Y 197.613,Z 742.661,A -85,B 0,C 180,E1 -21600,E2 -21600} C_VEL
LIN {X 0,Y 197.818,Z 747.003,A -85,B 0,C 180,E1 -21603.055,E2 -21603.055} C_VEL
LIN {X 0,Y 198.208,Z 750.317,A -85,B 0,C 180,E1 -21606.106,E2 -21606.106} C_VEL
LIN {X 0,Y 198.789,Z 752.042,A -85,B 0,C 180,E1 -21608.13,E2 -21608.13} C_VEL
LIN {X 0,Y 200.184,Z 753.771,A -85,B 0,C 180,E1 -21611.085,E2 -21611.085} C_VEL
LIN {X 0,Y 200.486,Z 754.482,A -85,B 0,C 180,E1 -21612.761,E2 -21612.761} C_VEL
LIN {X 0,Y 199.607,Z 755.172,A -85,B 0,C 180,E1 -21615.583,E2 -21615.583} C_VEL
LIN {X 0,Y 199.31,Z 755.385,A -85,B 0,C 180,E1 -21618.422,E2 -21618.422} C_VEL
LIN {X 0,Y 200.496,Z 755.13,A -85,B 0,C 180,E1 -21620.073,E2 -21620.073} C_VEL
LIN {X 0,Y 203.372,Z 754.335,A -85,B 0,C 180,E1 -21622.341,E2 -21622.341} C_VEL
LIN {X 0,Y 209.113,Z 751.728,A -85,B 0,C 180,E1 -21625.907,E2 -21625.907} C_VEL
LIN {X 0,Y 215.733,Z 747.568,A -85,B 0,C 180,E1 -21629.252,E2 -21629.252} C_VEL
LIN {X 0,Y 221.314,Z 743.333,A -85,B 0,C 180,E1 -21631.599,E2 -21631.599} C_VEL
LIN {X 0,Y 228.408,Z 737.112,A -85,B 0,C 180,E1 -21634.162,E2 -21634.162} C_VEL
LIN {X 0,Y 236.05,Z 729.253,A -85,B 0,C 180,E1 -21636.546,E2 -21636.546} C_VEL
LIN {X 0,Y 242.993,Z 721.066,A -85,B 0,C 180,E1 -21638.45,E2 -21638.45} C_VEL
LIN {X 0,Y 250.34,Z 711.165,A -85,B 0,C 180,E1 -21640.218,E2 -21640.218} C_VEL
LIN {X 0,Y 256.898,Z 700.986,A -85,B 0,C 180,E1 -21641.623,E2 -21641.623} C_VEL
LIN {X 0,Y 262.726,Z 690.417,A -85,B 0,C 180,E1 -21642.749,E2 -21642.749} C_VEL
LIN {X 0,Y 268.099,Z 679.005,A -85,B 0,C 180,E1 -21643.709,E2 -21643.709} C_VEL
LIN {X 0,Y 267.812,Z 679.603,A -85,B 0,C 180,E1 -21644.121,E2 -21644.121} C_VEL
LIN {X 0,Y 261.22,Z 693.183,A -85,B 0,C 180,E1 -21645.068,E2 -21645.068} C_VEL
LIN {X 0,Y 253.432,Z 706.576,A -85,B 0,C 180,E1 -21646.355,E2 -21646.355} C_VEL
LIN {X 0,Y 245.939,Z 717.707,A -85,B 0,C 180,E1 -21647.812,E2 -21647.812} C_VEL
LIN {X 0,Y 238.312,Z 727.752,A -85,B 0,C 180,E1 -21649.547,E2 -21649.547} C_VEL
LIN {X 0,Y 231.212,Z 736.162,A -85,B 0,C 180,E1 -21651.453,E2 -21651.453} C_VEL
LIN {X 0,Y 223.569,Z 744.35,A -85,B 0,C 180,E1 -21653.882,E2 -21653.882} C_VEL
LIN {X 0,Y 216.477,Z 751.186,A -85,B 0,C 180,E1 -21656.499,E2 -21656.499} C_VEL
LIN {X 0,Y 209.369,Z 757.391,A -85,B 0,C 180,E1 -21659.765,E2 -21659.765} C_VEL
LIN {X 0,Y 203.387,Z 762.01,A -85,B 0,C 180,E1 -21663.304,E2 -21663.304} C_VEL
LIN {X 0,Y 198.493,Z 765.257,A -85,B 0,C 180,E1 -21667.076,E2 -21667.076} C_VEL
LIN {X 0,Y 194.832,Z 767.17,A -85,B 0,C 180,E1 -21671.053,E2 -21671.053} C_VEL
LIN {X 0,Y 192.237,Z 767.704,A -85,B 0,C 180,E1 -21675.17,E2 -21675.17} C_VEL
LIN {X 0,Y 190.964,Z 766.855,A -85,B 0,C 180,E1 -21679.394,E2 -21679.394} C_VEL
LIN {X 0,Y 190.721,Z 765.932,A -85,B 0,C 180,E1 -21681.788,E2 -21681.788} C_VEL
LIN {X 0,Y 190.453,Z 767.979,A -85,B 0,C 180,E1 -21685.765,E2 -21685.765} C_VEL
LIN {X 0,Y 190.516,Z 768.552,A -85,B 0,C 180,E1 -21687.883,E2 -21687.883} C_VEL
LIN {X 0,Y 190.625,Z 768.747,A -85,B 0,C 180,E1 -21689.997,E2 -21689.997} C_VEL
LIN {X 0,Y 190.5,Z 768.54,A -85,B 0,C 180,E1 -21692.111,E2 -21692.111} C_VEL
LIN {X 0,Y 190.428,Z 767.726,A -85,B 0,C 180,E1 -21694.815,E2 -21694.815} C_VEL
LIN {X 0,Y 190.453,Z 765.683,A -85,B 0,C 180,E1 -21698.485,E2 -21698.485} C_VEL
LIN {X 0,Y 191.13,Z 761.887,A -85,B 0,C 180,E1 -21702.743,E2 -21702.743} C_VEL
LIN {X 0,Y 192.271,Z 757.961,A -85,B 0,C 180,E1 -21705.908,E2 -21705.908} C_VEL
LIN {X 0,Y 194.293,Z 751.556,A -85,B 0,C 180,E1 -21709.869,E2 -21709.869} C_VEL
LIN {X 0,Y 196.834,Z 744.726,A -85,B 0,C 180,E1 -21713.123,E2 -21713.123} C_VEL
LIN {X 0,Y 199.659,Z 736.927,A -85,B 0,C 180,E1 -21716.101,E2 -21716.101} C_VEL
LIN {X 0,Y 203.164,Z 727.499,A -85,B 0,C 180,E1 -21718.963,E2 -21718.963} C_VEL
LIN {X 0,Y 206.555,Z 717.334,A -85,B 0,C 180,E1 -21721.43,E2 -21721.43} C_VEL
LIN {X 0,Y 209.906,Z 706.46,A -85,B 0,C 180,E1 -21723.532,E2 -21723.532} C_VEL
LIN {X 0,Y 213.467,Z 693.587,A -85,B 0,C 180,E1 -21725.466,E2 -21725.466} C_VEL
LIN {X 0,Y 216.651,Z 679.903,A -85,B 0,C 180,E1 -21727.021,E2 -21727.021} C_VEL
LIN {X 0,Y 219.089,Z 666.446,A -85,B 0,C 180,E1 -21728.131,E2 -21728.131} C_VEL
LIN {X 0,Y 220.892,Z 652.474,A -85,B 0,C 180,E1 -21728.927,E2 -21728.927} C_VEL
LIN {X 0,Y 222.273,Z 631.997,A -85,B 0,C 180,E1 -21729.639,E2 -21729.639} C_VEL
LIN {X 0,Y 225.589,Z 573.413,A -85,B 0,C 180,E1 -21731.425,E2 -21731.425} C_VEL
LIN {X 0,Y 224.949,Z 566.969,A -85,B 0,C 180,E1 -21731.835,E2 -21731.835} C_VEL
LIN {X 0,Y 219.412,Z 554.214,A -85,B 0,C 180,E1 -21733.639,E2 -21733.639} C_VEL
LIN {X 0,Y 212.933,Z 541.407,A -85,B 0,C 180,E1 -21735.834,E2 -21735.834} C_VEL
LIN {X 0,Y 206.551,Z 530.151,A -85,B 0,C 180,E1 -21738.151,E2 -21738.151} C_VEL
LIN {X 0,Y 202.7,Z 524.215,A -85,B 0,C 180,E1 -21739.624,E2 -21739.624} C_VEL
LIN {X 0,Y 200.393,Z 520.313,A -85,B 0,C 180,E1 -21740.621,E2 -21740.621} C_VEL
LIN {X 0,Y 198.49,Z 514.164,A -85,B 0,C 180,E1 -21744.52,E2 -21744.52} C_VEL
LIN {X 0,Y 196.157,Z 507.671,A -85,B 0,C 180,E1 -21749.297,E2 -21749.297} C_VEL
LIN {X 0,Y 195.025,Z 504.331,A -85,B 0,C 180,E1 -21752.065,E2 -21752.065} C_VEL
LIN {X 0,Y 193.164,Z 499.92,A -85,B 0,C 180,E1 -21756.408,E2 -21756.408} C_VEL
LIN {X 0,Y 192.623,Z 498.065,A -85,B 0,C 180,E1 -21758.461,E2 -21758.461} C_VEL
LIN {X 0,Y 192.747,Z 498.092,A -85,B 0,C 180,E1 -21763.041,E2 -21763.041} C_VEL
LIN {X 0,Y 192.844,Z 498.081,A -85,B 0,C 180,E1 -21767.37,E2 -21767.37} C_VEL
LIN {X 0,Y 193.069,Z 498.058,A -85,B 0,C 180,E1 -21771.628,E2 -21771.628} C_VEL
LIN {X 0,Y 193.256,Z 498.022,A -85,B 0,C 180,E1 -21777.916,E2 -21777.916} C_VEL
LIN {X 0,Y 193.437,Z 498.006,A -85,B 0,C 180,E1 -21780,E2 -21780} C_VEL
LIN {X 0,Y 192.969,Z 498.057,A -85,B 0,C 180,E1 -21784.177,E2 -21784.177} C_VEL
LIN {X 0,Y 193.052,Z 498.046,A -85,B 0,C 180,E1 -21788.373,E2 -21788.373} C_VEL
LIN {X 0,Y 192.801,Z 498.08,A -85,B 0,C 180,E1 -21792.634,E2 -21792.634} C_VEL
LIN {X 0,Y 192.749,Z 498.09,A -85,B 0,C 180,E1 -21796.96,E2 -21796.96} C_VEL
LIN {X 0,Y 192.627,Z 498.106,A -85,B 0,C 180,E1 -21801.399,E2 -21801.399} C_VEL
LIN {X 0,Y 192.611,Z 498.111,A -85,B 0,C 180,E1 -21805.231,E2 -21805.231} C_VEL
LIN {X 0,Y 194.036,Z 502.292,A -85,B 0,C 180,E1 -21809.631,E2 -21809.631} C_VEL
LIN {X 0,Y 195.272,Z 505.546,A -85,B 0,C 180,E1 -21812.675,E2 -21812.675} C_VEL
LIN {X 0,Y 196.74,Z 509.644,A -85,B 0,C 180,E1 -21816.116,E2 -21816.116} C_VEL
LIN {X 0,Y 198.794,Z 516.185,A -85,B 0,C 180,E1 -21820.847,E2 -21820.847} C_VEL
LIN {X 0,Y 199.528,Z 518.575,A -85,B 0,C 180,E1 -21822.315,E2 -21822.315} C_VEL
LIN {X 0,Y 202.514,Z 523.195,A -85,B 0,C 180,E1 -21823.524,E2 -21823.524} C_VEL
LIN {X 0,Y 208.92,Z 533.471,A -85,B 0,C 180,E1 -21825.93,E2 -21825.93} C_VEL
LIN {X 0,Y 215.313,Z 545.084,A -85,B 0,C 180,E1 -21828.157,E2 -21828.157} C_VEL
LIN {X 0,Y 221.965,Z 559.009,A -85,B 0,C 180,E1 -21830.327,E2 -21830.327} C_VEL
LIN {X 0,Y 224.485,Z 565.098,A -85,B 0,C 180,E1 -21831.128,E2 -21831.128} C_VEL
LIN {X 0,Y 225.262,Z 571.199,A -85,B 0,C 180,E1 -21831.535,E2 -21831.535} C_VEL
LIN {X 0,Y 221.901,Z 636.907,A -85,B 0,C 180,E1 -21833.432,E2 -21833.432} C_VEL
LIN {X 0,Y 220.616,Z 649.703,A -85,B 0,C 180,E1 -21834.105,E2 -21834.105} C_VEL
LIN {X 0,Y 218.757,Z 662.314,A -85,B 0,C 180,E1 -21835.095,E2 -21835.095} C_VEL
LIN {X 0,Y 216.621,Z 673.268,A -85,B 0,C 180,E1 -21836.251,E2 -21836.251} C_VEL
LIN {X 0,Y 213.522,Z 685.689,A -85,B 0,C 180,E1 -21837.947,E2 -21837.947} C_VEL
LIN {X 0,Y 210.271,Z 696.724,A -85,B 0,C 180,E1 -21839.914,E2 -21839.914} C_VEL
LIN {X 0,Y 207.231,Z 706.124,A -85,B 0,C 180,E1 -21842.056,E2 -21842.056} C_VEL
LIN {X 0,Y 204.024,Z 714.79,A -85,B 0,C 180,E1 -21844.498,E2 -21844.498} C_VEL
LIN {X 0,Y 200.752,Z 722.861,A -85,B 0,C 180,E1 -21847.354,E2 -21847.354} C_VEL
LIN {X 0,Y 198.047,Z 729.419,A -85,B 0,C 180,E1 -21850.301,E2 -21850.301} C_VEL
LIN {X 0,Y 195.72,Z 734.724,A -85,B 0,C 180,E1 -21853.309,E2 -21853.309} C_VEL
LIN {X 0,Y 193.789,Z 738.948,A -85,B 0,C 180,E1 -21856.368,E2 -21856.368} C_VEL
LIN {X 0,Y 192.454,Z 742.192,A -85,B 0,C 180,E1 -21859.482,E2 -21859.482} C_VEL
LIN {X 0,Y 191.343,Z 745.085,A -85,B 0,C 180,E1 -21863.677,E2 -21863.677} C_VEL
LIN {X 0,Y 190.754,Z 746.541,A -85,B 0,C 180,E1 -21867.891,E2 -21867.891} C_VEL
LIN {X 0,Y 190.753,Z 746.572,A -85,B 0,C 180,E1 -21872.114,E2 -21872.114} C_VEL
LIN {X 0,Y 191.337,Z 745.154,A -85,B 0,C 180,E1 -21876.329,E2 -21876.329} C_VEL
LIN {X 0,Y 192.458,Z 742.303,A -85,B 0,C 180,E1 -21880.523,E2 -21880.523} C_VEL
LIN {X 0,Y 193.788,Z 739.108,A -85,B 0,C 180,E1 -21883.637,E2 -21883.637} C_VEL
LIN {X 0,Y 195.685,Z 734.936,A -85,B 0,C 180,E1 -21886.7,E2 -21886.7} C_VEL
LIN {X 0,Y 197.968,Z 729.684,A -85,B 0,C 180,E1 -21889.712,E2 -21889.712} C_VEL
LIN {X 0,Y 201.236,Z 721.976,A -85,B 0,C 180,E1 -21893.137,E2 -21893.137} C_VEL
LIN {X 0,Y 204.597,Z 713.699,A -85,B 0,C 180,E1 -21895.977,E2 -21895.977} C_VEL
LIN {X 0,Y 207.691,Z 704.955,A -85,B 0,C 180,E1 -21898.38,E2 -21898.38} C_VEL
